// SIMATIC STEP 7 (V5.x) project Daysil_Autoklv_v3_upload
// station: P_ADR_BUS
// station: Hardware
// station: SLIO_CPU_015
// program: S7 Program(1)

FUNCTION_BLOCK FB 1
VERSION : 0.1
BEGIN
// (block stored without names or comments; labels and parameter names are numbered)
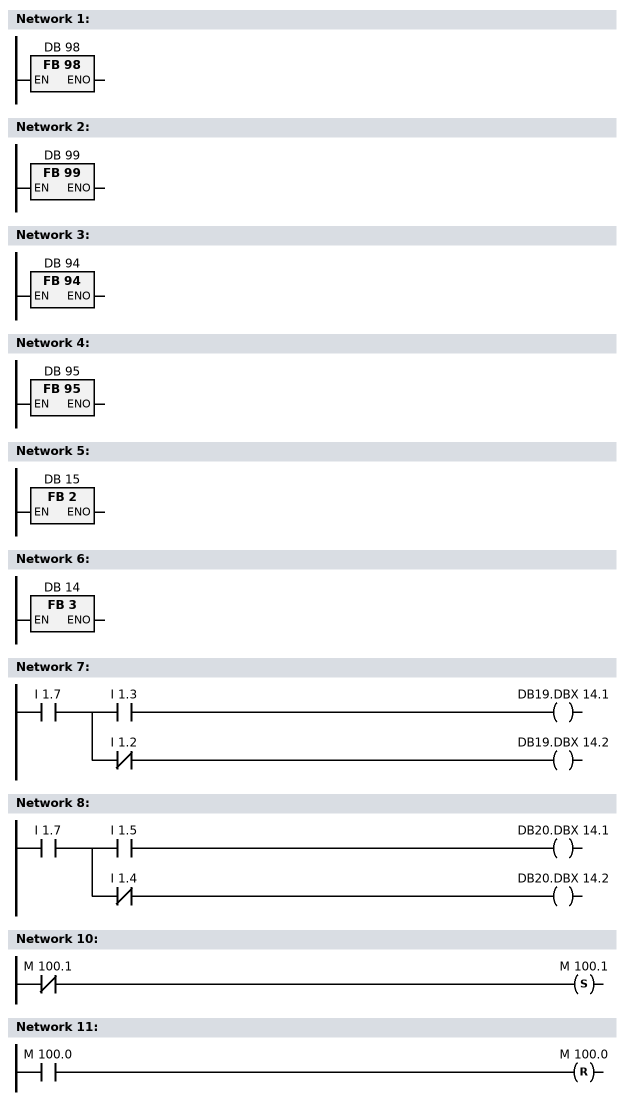
NETWORK
TITLE =
      CALL  FB 98 , DB 98;
      NOP   0;
NETWORK
TITLE =
      CALL  FB 99 , DB 99;
      NOP   0;
NETWORK
TITLE =
      CALL  FB 94 , DB 94;
      NOP   0;
NETWORK
TITLE =
      CALL  FB 95 , DB 95;
      NOP   0;
NETWORK
TITLE =
      CALL  FB 2 , DB 15;
      NOP   0;
NETWORK
TITLE =
      CALL  FB 3 , DB 14;
      NOP   0;
NETWORK
TITLE =
      A     I 1.7;
      =     L 0.0;
      A     L 0.0;
      A     I 1.3;
      =     DB19.DBX 14.1;
      A     L 0.0;
      AN    I 1.2;
      =     DB19.DBX 14.2;
NETWORK
TITLE =
      A     I 1.7;
      =     L 0.0;
      A     L 0.0;
      A     I 1.5;
      =     DB20.DBX 14.1;
      A     L 0.0;
      AN    I 1.4;
      =     DB20.DBX 14.2;
NETWORK
TITLE =
NETWORK
TITLE =
      AN    M 100.1;
      S     M 100.1;
NETWORK
TITLE =
      A     M 100.0;
      R     M 100.0;
NETWORK
TITLE =
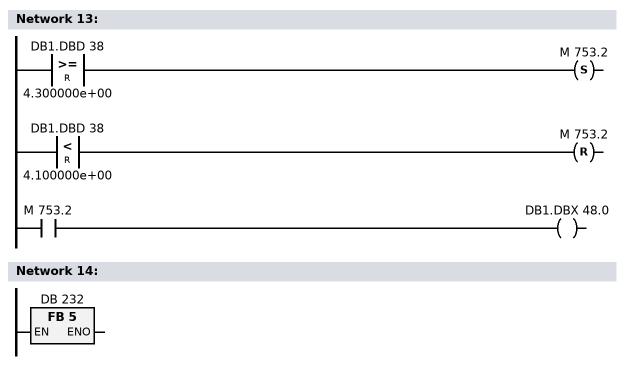
NETWORK
TITLE =
      A(;
      L     DB1.DBD 38;
      L     4.300000e+00;
      >=R;
      );
      S     M 753.2;
      A(;
      L     DB1.DBD 38;
      L     4.100000e+00;
      <R;
      );
      R     M 753.2;
      A     M 753.2;
      =     DB1.DBX 48.0;
NETWORK
TITLE =
      CALL  FB 5 , DB 232;
      NOP   0;
END_FUNCTION_BLOCK

FUNCTION_BLOCK FB 2
VERSION : 0.1
BEGIN
// (block stored without names or comments; labels and parameter names are numbered)
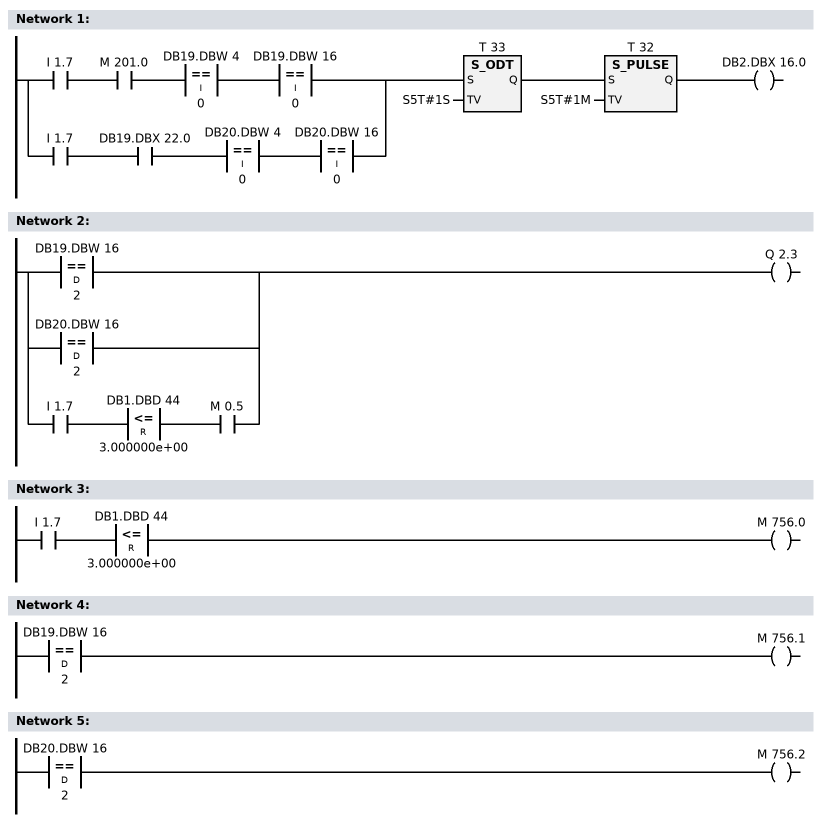
NETWORK
TITLE =
      A(;
      A(;
      A     I 1.7;
      A     M 201.0;
      A(;
      L     DB19.DBW 4;
      L     0;
      ==I;
      );
      A(;
      L     DB19.DBW 16;
      L     0;
      ==I;
      );
      O;
      A     I 1.7;
      A     DB19.DBX 22.0;
      A(;
      L     DB20.DBW 4;
      L     0;
      ==I;
      );
      A(;
      L     DB20.DBW 16;
      L     0;
      ==I;
      );
      );
      L     S5T#1S;
      SD    T 33;
      NOP   0;
      NOP   0;
      NOP   0;
      A     T 33;
      );
      L     S5T#1M;
      SP    T 32;
      NOP   0;
      NOP   0;
      NOP   0;
      A     T 32;
      =     DB2.DBX 16.0;
NETWORK
TITLE =
      O(;
      L     DB19.DBW 16;
      L     2;
      ==D;
      );
      O(;
      L     DB20.DBW 16;
      L     2;
      ==D;
      );
      O;
      A     I 1.7;
      A(;
      L     DB1.DBD 44;
      L     3.000000e+00;
      <=R;
      );
      A     M 0.5;
      =     Q 2.3;
NETWORK
TITLE =
      A     I 1.7;
      A(;
      L     DB1.DBD 44;
      L     3.000000e+00;
      <=R;
      );
      =     M 756.0;
NETWORK
TITLE =
      L     DB19.DBW 16;
      L     2;
      ==D;
      =     M 756.1;
NETWORK
TITLE =
      L     DB20.DBW 16;
      L     2;
      ==D;
      =     M 756.2;
END_FUNCTION_BLOCK

FUNCTION_BLOCK FB 3
VERSION : 0.1
BEGIN
// (block stored without names or comments; labels and parameter names are numbered)
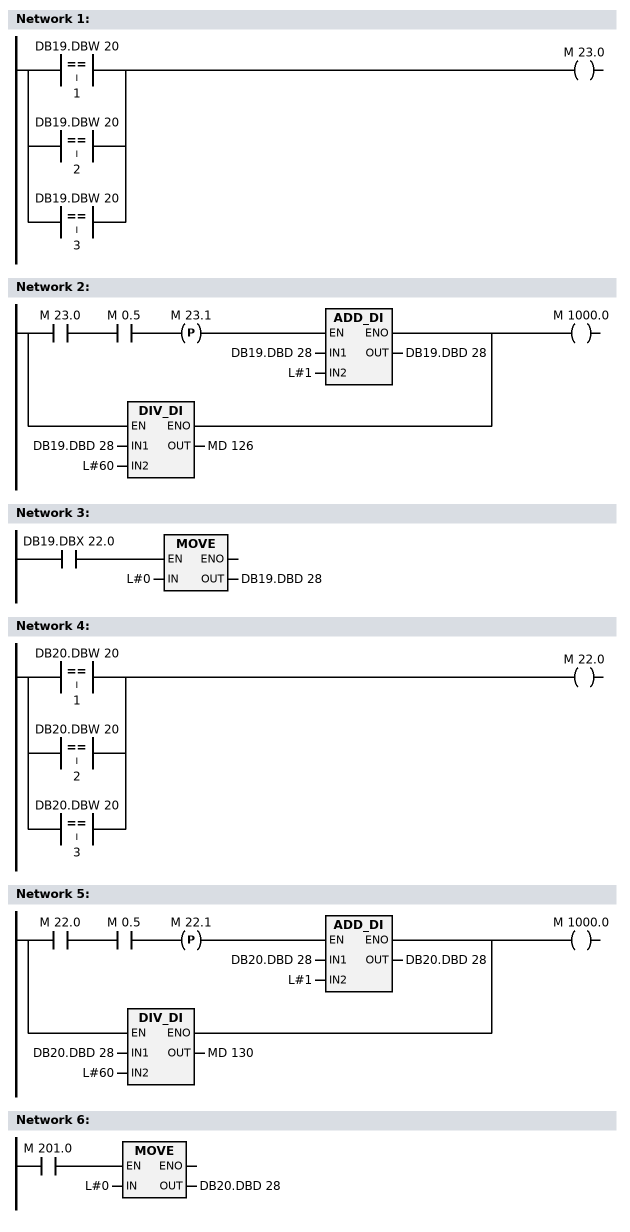
NETWORK
TITLE =
      O(;
      L     DB19.DBW 20;
      L     1;
      ==I;
      );
      O(;
      L     DB19.DBW 20;
      L     2;
      ==I;
      );
      O(;
      L     DB19.DBW 20;
      L     3;
      ==I;
      );
      =     M 23.0;
NETWORK
TITLE =
      O(;
      A     M 23.0;
      A     M 0.5;
      FP    M 23.1;
      JNB   M001;
      L     DB19.DBD 28;
      L     L#1;
      +D;
      T     DB19.DBD 28;
      AN    OV;
      SAVE;
      CLR;
M001: A     BR;
      );
      O(;
      L     DB19.DBD 28;
      L     L#60;
      /D;
      T     MD 126;
      AN    OV;
      SAVE;
      CLR;
      A     BR;
      );
      =     M 1000.0;
NETWORK
TITLE =
      A     DB19.DBX 22.0;
      JNB   M002;
      L     L#0;
      T     DB19.DBD 28;
M002: NOP   0;
NETWORK
TITLE =
      O(;
      L     DB20.DBW 20;
      L     1;
      ==I;
      );
      O(;
      L     DB20.DBW 20;
      L     2;
      ==I;
      );
      O(;
      L     DB20.DBW 20;
      L     3;
      ==I;
      );
      =     M 22.0;
NETWORK
TITLE =
      O(;
      A     M 22.0;
      A     M 0.5;
      FP    M 22.1;
      JNB   M003;
      L     DB20.DBD 28;
      L     L#1;
      +D;
      T     DB20.DBD 28;
      AN    OV;
      SAVE;
      CLR;
M003: A     BR;
      );
      O(;
      L     DB20.DBD 28;
      L     L#60;
      /D;
      T     MD 130;
      AN    OV;
      SAVE;
      CLR;
      A     BR;
      );
      =     M 1000.0;
NETWORK
TITLE =
      A     M 201.0;
      JNB   M004;
      L     L#0;
      T     DB20.DBD 28;
M004: NOP   0;
NETWORK
TITLE =
      O(;
      A(;
      A     DB17.DBX 40.3;
      =     L 0.0;
      BLD   103;
      BLD   9;
      =     L 5.0;
      CDB;
      OPN   DI 5;
      TAR2  LD 1;
      A     L 0.0;
      =     DIX 0.0;
      L     L#82800000;
      T     DID 2;
      LAR2  P#DBX 0.0;
      UC    SFB 4;
      LAR2  LD 1;
      L     DID 8;
      OPN   DI 17;
      T     DID 42;
      OPN   DI 5;
      CDB;
      BLD   10;
      A     BR;
      );
      JNB   M005;
      CALL  FC 1 (
           $1                       := DB17.DBD 42,
           $2                       := DB17.DBW 4,
           $3                       := DB17.DBD 46);
M005: A     BR;
      );
      O(;
      L     DB17.DBD 46;
      L     60;
      /D;
      T     MD 118;
      AN    OV;
      SAVE;
      CLR;
      A     BR;
      );
      =     M 1000.0;
NETWORK
TITLE =
      O(;
      A(;
      A     DB18.DBX 40.3;
      =     L 0.0;
      BLD   103;
      BLD   9;
      =     L 5.0;
      CDB;
      OPN   DI 6;
      TAR2  LD 1;
      A     L 0.0;
      =     DIX 0.0;
      L     L#82800000;
      T     DID 2;
      LAR2  P#DBX 0.0;
      UC    SFB 4;
      LAR2  LD 1;
      L     DID 8;
      OPN   DI 18;
      T     DID 42;
      OPN   DI 6;
      CDB;
      BLD   10;
      A     BR;
      );
      JNB   M006;
      CALL  FC 1 (
           $1                       := DB18.DBD 42,
           $2                       := DB18.DBW 4,
           $3                       := DB18.DBD 46);
M006: A     BR;
      );
      O(;
      L     DB18.DBD 46;
      L     60;
      /D;
      T     MD 122;
      AN    OV;
      SAVE;
      CLR;
      A     BR;
      );
      =     M 1000.0;
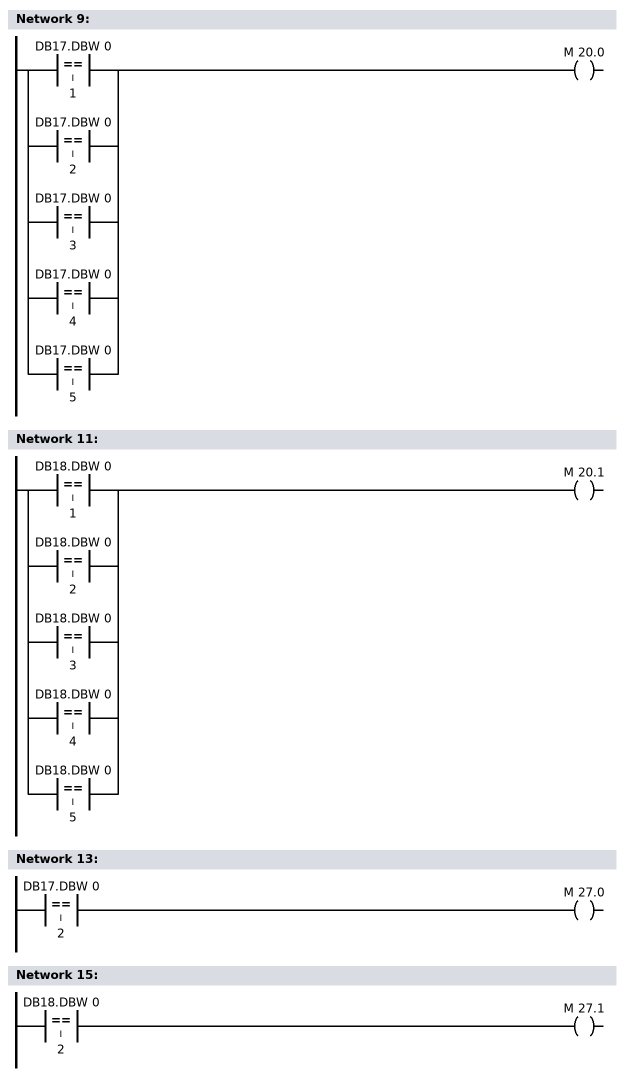
NETWORK
TITLE =
      O(;
      L     DB17.DBW 0;
      L     1;
      ==I;
      );
      O(;
      L     DB17.DBW 0;
      L     2;
      ==I;
      );
      O(;
      L     DB17.DBW 0;
      L     3;
      ==I;
      );
      O(;
      L     DB17.DBW 0;
      L     4;
      ==I;
      );
      O(;
      L     DB17.DBW 0;
      L     5;
      ==I;
      );
      =     M 20.0;
NETWORK
TITLE =
      O(;
      A(;
      A     M 20.0;
      =     L 0.0;
      BLD   103;
      BLD   9;
      =     L 5.0;
      CDB;
      OPN   DI 7;
      TAR2  LD 1;
      A     L 0.0;
      =     DIX 0.0;
      L     L#82800000;
      T     DID 2;
      LAR2  P#DBX 0.0;
      UC    SFB 4;
      LAR2  LD 1;
      L     DID 8;
      OPN   DI 17;
      T     DID 50;
      OPN   DI 7;
      CDB;
      BLD   10;
      A     BR;
      );
      JNB   M007;
      L     DB17.DBD 50;
      L     1000;
      /D;
      T     DB17.DBD 54;
      AN    OV;
      SAVE;
      CLR;
M007: A     BR;
      );
      O(;
      L     DB17.DBD 54;
      L     60;
      /D;
      T     MD 110;
      AN    OV;
      SAVE;
      CLR;
      A     BR;
      );
      =     M 1000.0;
NETWORK
TITLE =
      O(;
      L     DB18.DBW 0;
      L     1;
      ==I;
      );
      O(;
      L     DB18.DBW 0;
      L     2;
      ==I;
      );
      O(;
      L     DB18.DBW 0;
      L     3;
      ==I;
      );
      O(;
      L     DB18.DBW 0;
      L     4;
      ==I;
      );
      O(;
      L     DB18.DBW 0;
      L     5;
      ==I;
      );
      =     M 20.1;
NETWORK
TITLE =
      O(;
      A(;
      A     M 20.1;
      =     L 0.0;
      BLD   103;
      BLD   9;
      =     L 5.0;
      CDB;
      OPN   DI 8;
      TAR2  LD 1;
      A     L 0.0;
      =     DIX 0.0;
      L     L#82800000;
      T     DID 2;
      LAR2  P#DBX 0.0;
      UC    SFB 4;
      LAR2  LD 1;
      L     DID 8;
      OPN   DI 18;
      T     DID 50;
      OPN   DI 8;
      CDB;
      BLD   10;
      A     BR;
      );
      JNB   M008;
      L     DB18.DBD 50;
      L     1000;
      /D;
      T     DB18.DBD 54;
      AN    OV;
      SAVE;
      CLR;
M008: A     BR;
      );
      O(;
      L     DB18.DBD 54;
      L     60;
      /D;
      T     MD 114;
      AN    OV;
      SAVE;
      CLR;
      A     BR;
      );
      =     M 1000.0;
NETWORK
TITLE =
      L     DB17.DBW 0;
      L     2;
      ==I;
      =     M 27.0;
NETWORK
TITLE =
      A(;
      A     M 27.0;
      =     L 0.0;
      BLD   103;
      BLD   9;
      =     L 5.0;
      CDB;
      OPN   DI 9;
      TAR2  LD 1;
      A     L 0.0;
      =     DIX 0.0;
      L     L#82800000;
      T     DID 2;
      LAR2  P#DBX 0.0;
      UC    SFB 4;
      LAR2  LD 1;
      L     DID 8;
      OPN   DI 17;
      T     DID 58;
      OPN   DI 9;
      CDB;
      BLD   10;
      A     BR;
      );
      JNB   M009;
      L     DB17.DBD 58;
      L     1000;
      /D;
      T     DB17.DBD 62;
M009: NOP   0;
NETWORK
TITLE =
      L     DB18.DBW 0;
      L     2;
      ==I;
      =     M 27.1;
NETWORK
TITLE =
      A(;
      A     M 27.1;
      =     L 0.0;
      BLD   103;
      BLD   9;
      =     L 5.0;
      CDB;
      OPN   DI 10;
      TAR2  LD 1;
      A     L 0.0;
      =     DIX 0.0;
      L     L#82800000;
      T     DID 2;
      LAR2  P#DBX 0.0;
      UC    SFB 4;
      LAR2  LD 1;
      L     DID 8;
      OPN   DI 18;
      T     DID 58;
      OPN   DI 10;
      CDB;
      BLD   10;
      A     BR;
      );
      JNB   M010;
      L     DB18.DBD 58;
      L     1000;
      /D;
      T     DB18.DBD 62;
M010: NOP   0;
END_FUNCTION_BLOCK

FUNCTION_BLOCK FB 5
VERSION : 0.1
BEGIN
// (block stored without names or comments; labels and parameter names are numbered)
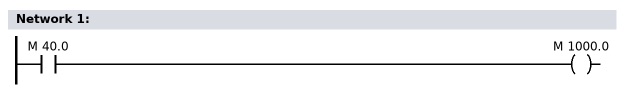
NETWORK
TITLE =
      A     M 40.0;
      =     M 1000.0;
END_FUNCTION_BLOCK

FUNCTION_BLOCK FB 20
VERSION : 0.1
BEGIN
// (block stored without names or comments; labels and parameter names are numbered)
NETWORK
TITLE =
      A(;
      A(;
      A     M 100.0;
      =     L 0.0;
      BLD   103;
      CALL  FC 105 (
           $1                       := DIW [AR2,P#4.0],
           $2                       := DID [AR2,P#24.0],
           $3                       := DID [AR2,P#28.0],
           $4                       := L 0.0,
           $5                       := DIW [AR2,P#116.0],
           $6                       := DID [AR2,P#118.0]);
      A     BR;
      );
      JNB   M001;
      L     DIW [AR2,P#116.0];
      T     DIW [AR2,P#68.0];
      SET;
      SAVE;
      CLR;
M001: A     BR;
      );
      JNB   M002;
      L     DID [AR2,P#118.0];
      T     DID [AR2,P#70.0];
M002: NOP   0;
NETWORK
TITLE =
      A(;
      A(;
      A     M 100.0;
      =     L 0.0;
      BLD   103;
      CALL  FC 105 (
           $1                       := DIW [AR2,P#40.0],
           $2                       := DID [AR2,P#32.0],
           $3                       := DID [AR2,P#36.0],
           $4                       := L 0.0,
           $5                       := DIW [AR2,P#122.0],
           $6                       := DID [AR2,P#124.0]);
      A     BR;
      );
      JNB   M003;
      L     DIW [AR2,P#122.0];
      T     DIW [AR2,P#76.0];
      SET;
      SAVE;
      CLR;
M003: A     BR;
      );
      JNB   M004;
      L     DID [AR2,P#124.0];
      T     DID [AR2,P#78.0];
M004: NOP   0;
NETWORK
TITLE =
      A(;
      A     I 1.7;
      A     DIX [AR2,P#0.0];
      A     DB1.DBX 48.0;
      L     S5T#200MS;
      T     LD 0;
      TAK;
      T     LD 4;
      L     DIW [AR2,P#14.0];
      T     LW 8;
      L     LD 4;
      L     LD 0;
      SD    T [LW 8];
      NOP   0;
      NOP   0;
      NOP   0;
      T     LD 0;
      TAK;
      T     LD 4;
      L     DIW [AR2,P#14.0];
      T     LW 8;
      L     LD 4;
      L     LD 0;
      A     T [LW 8];
      );
      A     DIX [AR2,P#0.4];
      A     DIX [AR2,P#0.1];
      A(;
      L     DIW [AR2,P#84.0];
      L     0;
      ==I;
      );
      JNB   M005;
      L     1;
      T     DIW [AR2,P#84.0];
      SET;
      SAVE;
      CLR;
M005: A     BR;
      S     DIX [AR2,P#128.0];
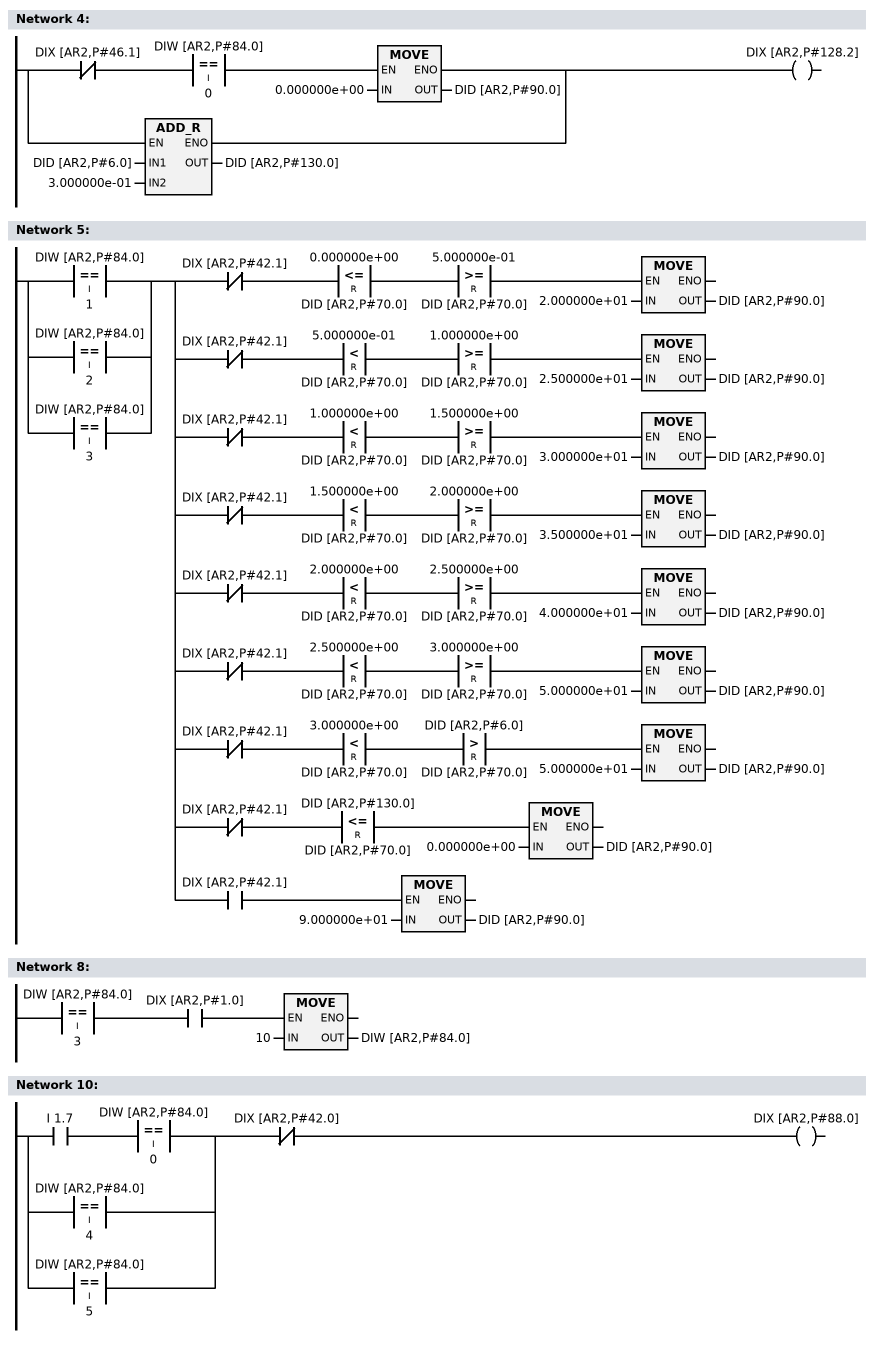
NETWORK
TITLE =
      O(;
      AN    DIX [AR2,P#46.1];
      A(;
      L     DIW [AR2,P#84.0];
      L     0;
      ==I;
      );
      JNB   M006;
      L     0.000000e+00;
      T     DID [AR2,P#90.0];
      SET;
      SAVE;
      CLR;
M006: A     BR;
      );
      O(;
      L     DID [AR2,P#6.0];
      L     3.000000e-01;
      +R;
      T     DID [AR2,P#130.0];
      AN    OV;
      SAVE;
      CLR;
      A     BR;
      );
      =     DIX [AR2,P#128.2];
NETWORK
TITLE =
      O(;
      L     DIW [AR2,P#84.0];
      L     1;
      ==I;
      );
      O(;
      L     DIW [AR2,P#84.0];
      L     2;
      ==I;
      );
      O(;
      L     DIW [AR2,P#84.0];
      L     3;
      ==I;
      );
      =     L 0.0;
      A     L 0.0;
      AN    DIX [AR2,P#42.1];
      A(;
      L     0.000000e+00;
      L     DID [AR2,P#70.0];
      <=R;
      );
      A(;
      L     5.000000e-01;
      L     DID [AR2,P#70.0];
      >=R;
      );
      JNB   M007;
      L     2.000000e+01;
      T     DID [AR2,P#90.0];
M007: NOP   0;
      A     L 0.0;
      AN    DIX [AR2,P#42.1];
      A(;
      L     5.000000e-01;
      L     DID [AR2,P#70.0];
      <R;
      );
      A(;
      L     1.000000e+00;
      L     DID [AR2,P#70.0];
      >=R;
      );
      JNB   M008;
      L     2.500000e+01;
      T     DID [AR2,P#90.0];
M008: NOP   0;
      A     L 0.0;
      AN    DIX [AR2,P#42.1];
      A(;
      L     1.000000e+00;
      L     DID [AR2,P#70.0];
      <R;
      );
      A(;
      L     1.500000e+00;
      L     DID [AR2,P#70.0];
      >=R;
      );
      JNB   M009;
      L     3.000000e+01;
      T     DID [AR2,P#90.0];
M009: NOP   0;
      A     L 0.0;
      AN    DIX [AR2,P#42.1];
      A(;
      L     1.500000e+00;
      L     DID [AR2,P#70.0];
      <R;
      );
      A(;
      L     2.000000e+00;
      L     DID [AR2,P#70.0];
      >=R;
      );
      JNB   M010;
      L     3.500000e+01;
      T     DID [AR2,P#90.0];
M010: NOP   0;
      A     L 0.0;
      AN    DIX [AR2,P#42.1];
      A(;
      L     2.000000e+00;
      L     DID [AR2,P#70.0];
      <R;
      );
      A(;
      L     2.500000e+00;
      L     DID [AR2,P#70.0];
      >=R;
      );
      JNB   M011;
      L     4.000000e+01;
      T     DID [AR2,P#90.0];
M011: NOP   0;
      A     L 0.0;
      AN    DIX [AR2,P#42.1];
      A(;
      L     2.500000e+00;
      L     DID [AR2,P#70.0];
      <R;
      );
      A(;
      L     3.000000e+00;
      L     DID [AR2,P#70.0];
      >=R;
      );
      JNB   M012;
      L     5.000000e+01;
      T     DID [AR2,P#90.0];
M012: NOP   0;
      A     L 0.0;
      AN    DIX [AR2,P#42.1];
      A(;
      L     3.000000e+00;
      L     DID [AR2,P#70.0];
      <R;
      );
      A(;
      L     DID [AR2,P#6.0];
      L     DID [AR2,P#70.0];
      >R;
      );
      JNB   M013;
      L     5.000000e+01;
      T     DID [AR2,P#90.0];
M013: NOP   0;
      A     L 0.0;
      AN    DIX [AR2,P#42.1];
      A(;
      L     DID [AR2,P#130.0];
      L     DID [AR2,P#70.0];
      <=R;
      );
      JNB   M014;
      L     0.000000e+00;
      T     DID [AR2,P#90.0];
M014: NOP   0;
      A     L 0.0;
      A     DIX [AR2,P#42.1];
      JNB   M015;
      L     9.000000e+01;
      T     DID [AR2,P#90.0];
M015: NOP   0;
NETWORK
TITLE =
      L     DIW [AR2,P#84.0];
      L     1;
      ==I;
      =     L 0.0;
      A(;
      A     L 0.0;
      A     DIX [AR2,P#104.0];
      L     DIW [AR2,P#2.0];
      T     LD 1;
      TAK;
      T     LD 5;
      L     DIW [AR2,P#18.0];
      T     LW 9;
      L     LD 5;
      L     LD 1;
      SD    T [LW 9];
      NOP   0;
      NOP   0;
      NOP   0;
      T     LD 1;
      TAK;
      T     LD 5;
      L     DIW [AR2,P#18.0];
      T     LW 9;
      L     LD 5;
      L     LD 1;
      A     T [LW 9];
      );
      JNB   M016;
      L     2;
      T     DIW [AR2,P#84.0];
M016: NOP   0;
      A     L 0.0;
      A(;
      O(;
      L     DID [AR2,P#70.0];
      L     DID [AR2,P#6.0];
      >=R;
      );
      O     DIX [AR2,P#104.0];
      );
      =     DIX [AR2,P#104.0];
NETWORK
TITLE =
      L     DIW [AR2,P#84.0];
      L     2;
      ==I;
      =     L 0.0;
      A     L 0.0;
      L     S5T#5M;
      T     LD 1;
      TAK;
      T     LD 5;
      L     DIW [AR2,P#56.0];
      T     LW 9;
      L     LD 5;
      L     LD 1;
      SD    T [LW 9];
      NOP   0;
      NOP   0;
      NOP   0;
      NOP   0;
      A     L 0.0;
      A     DIX [AR2,P#0.2];
      JNB   M017;
      L     3;
      T     DIW [AR2,P#84.0];
M017: NOP   0;
      A     L 0.0;
      A     DIX [AR2,P#0.3];
      JNB   M018;
      L     4;
      T     DIW [AR2,P#84.0];
M018: NOP   0;
NETWORK
TITLE =
      A(;
      L     DIW [AR2,P#84.0];
      L     3;
      ==I;
      );
      A     DIX [AR2,P#1.0];
      JNB   M019;
      L     10;
      T     DIW [AR2,P#84.0];
M019: NOP   0;
NETWORK
TITLE =
      L     DIW [AR2,P#84.0];
      L     10;
      ==I;
      =     L 0.0;
      A     L 0.0;
      JNB   M020;
      L     9.000000e+01;
      T     DID [AR2,P#90.0];
      SET;
      SAVE;
      CLR;
M020: A     BR;
      =     DIX [AR2,P#66.0];
      A(;
      A     L 0.0;
      L     S5T#23S;
      T     LD 1;
      TAK;
      T     LD 5;
      L     DIW [AR2,P#20.0];
      T     LW 9;
      L     LD 5;
      L     LD 1;
      SD    T [LW 9];
      NOP   0;
      NOP   0;
      NOP   0;
      T     LD 1;
      TAK;
      T     LD 5;
      L     DIW [AR2,P#20.0];
      T     LW 9;
      L     LD 5;
      L     LD 1;
      A     T [LW 9];
      );
      JNB   M021;
      L     4;
      T     DIW [AR2,P#84.0];
M021: NOP   0;
NETWORK
TITLE =
      A(;
      A     I 1.7;
      A(;
      L     DIW [AR2,P#84.0];
      L     0;
      ==I;
      );
      O(;
      L     DIW [AR2,P#84.0];
      L     4;
      ==I;
      );
      O(;
      L     DIW [AR2,P#84.0];
      L     5;
      ==I;
      );
      );
      AN    DIX [AR2,P#42.0];
      =     DIX [AR2,P#88.0];
NETWORK
TITLE =
      L     DIW [AR2,P#84.0];
      L     4;
      ==I;
      =     L 0.0;
      A     L 0.0;
      JNB   M022;
      L     0.000000e+00;
      T     DID [AR2,P#90.0];
M022: NOP   0;
      A     L 0.0;
      BLD   102;
      =     DIX [AR2,P#128.1];
      A     L 0.0;
      A(;
      L     DID [AR2,P#70.0];
      L     1.000000e-01;
      <=R;
      );
      =     L 0.1;
      A     L 0.1;
      BLD   102;
      S     DIX [AR2,P#114.1];
      A(;
      A     L 0.1;
      L     S5T#5S;
      T     LD 1;
      TAK;
      T     LD 5;
      L     DIW [AR2,P#52.0];
      T     LW 9;
      L     LD 5;
      L     LD 1;
      SD    T [LW 9];
      NOP   0;
      NOP   0;
      NOP   0;
      T     LD 1;
      TAK;
      T     LD 5;
      L     DIW [AR2,P#52.0];
      T     LW 9;
      L     LD 5;
      L     LD 1;
      A     T [LW 9];
      );
      JNB   M023;
      L     5;
      T     DIW [AR2,P#84.0];
M023: NOP   0;
NETWORK
TITLE =
      A(;
      A(;
      L     DIW [AR2,P#84.0];
      L     5;
      ==I;
      );
      L     S5T#1S;
      T     LD 0;
      TAK;
      T     LD 4;
      L     DIW [AR2,P#54.0];
      T     LW 8;
      L     LD 4;
      L     LD 0;
      SD    T [LW 8];
      NOP   0;
      NOP   0;
      NOP   0;
      T     LD 0;
      TAK;
      T     LD 4;
      L     DIW [AR2,P#54.0];
      T     LW 8;
      L     LD 4;
      L     LD 0;
      A     T [LW 8];
      );
      AN    DIX [AR2,P#0.4];
      JNB   M024;
      L     0;
      T     DIW [AR2,P#84.0];
M024: NOP   0;
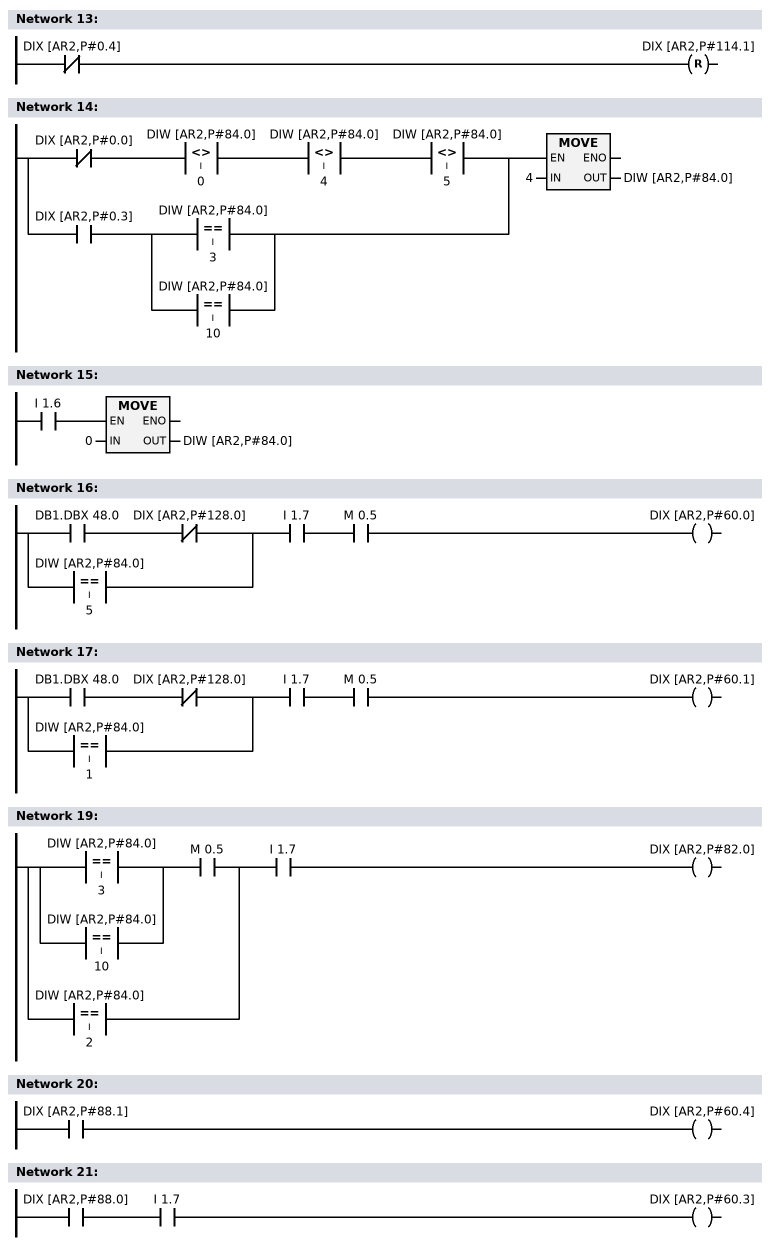
NETWORK
TITLE =
      AN    DIX [AR2,P#0.4];
      R     DIX [AR2,P#114.1];
NETWORK
TITLE =
      A(;
      AN    DIX [AR2,P#0.0];
      A(;
      L     DIW [AR2,P#84.0];
      L     0;
      <>I;
      );
      A(;
      L     DIW [AR2,P#84.0];
      L     4;
      <>I;
      );
      A(;
      L     DIW [AR2,P#84.0];
      L     5;
      <>I;
      );
      O;
      A     DIX [AR2,P#0.3];
      A(;
      O(;
      L     DIW [AR2,P#84.0];
      L     3;
      ==I;
      );
      O(;
      L     DIW [AR2,P#84.0];
      L     10;
      ==I;
      );
      );
      );
      JNB   M025;
      L     4;
      T     DIW [AR2,P#84.0];
M025: NOP   0;
NETWORK
TITLE =
      A     I 1.6;
      JNB   M026;
      L     0;
      T     DIW [AR2,P#84.0];
M026: NOP   0;
NETWORK
TITLE =
      A(;
      A     DB1.DBX 48.0;
      AN    DIX [AR2,P#128.0];
      O(;
      L     DIW [AR2,P#84.0];
      L     5;
      ==I;
      );
      );
      A     I 1.7;
      A     M 0.5;
      =     DIX [AR2,P#60.0];
NETWORK
TITLE =
      A(;
      A     DB1.DBX 48.0;
      AN    DIX [AR2,P#128.0];
      O(;
      L     DIW [AR2,P#84.0];
      L     1;
      ==I;
      );
      );
      A     I 1.7;
      A     M 0.5;
      =     DIX [AR2,P#60.1];
NETWORK
TITLE =
      A(;
      A(;
      L     DIW [AR2,P#84.0];
      L     2;
      ==I;
      );
      A     M 0.5;
      O(;
      A(;
      O(;
      L     DIW [AR2,P#84.0];
      L     3;
      ==I;
      );
      O(;
      L     DIW [AR2,P#84.0];
      L     10;
      ==I;
      );
      );
      AN    DIX [AR2,P#66.0];
      L     S5T#5M;
      T     LD 0;
      TAK;
      T     LD 4;
      L     DIW [AR2,P#58.0];
      T     LW 8;
      L     LD 4;
      L     LD 0;
      SD    T [LW 8];
      NOP   0;
      NOP   0;
      NOP   0;
      T     LD 0;
      TAK;
      T     LD 4;
      L     DIW [AR2,P#58.0];
      T     LW 8;
      L     LD 4;
      L     LD 0;
      A     T [LW 8];
      );
      );
      A     I 1.7;
      =     DIX [AR2,P#60.2];
NETWORK
TITLE =
      A(;
      A(;
      O(;
      L     DIW [AR2,P#84.0];
      L     3;
      ==I;
      );
      O(;
      L     DIW [AR2,P#84.0];
      L     10;
      ==I;
      );
      );
      A     M 0.5;
      O(;
      L     DIW [AR2,P#84.0];
      L     2;
      ==I;
      );
      );
      A     I 1.7;
      =     DIX [AR2,P#82.0];
NETWORK
TITLE =
      A     DIX [AR2,P#88.1];
      =     DIX [AR2,P#60.4];
NETWORK
TITLE =
      A     DIX [AR2,P#88.0];
      A     I 1.7;
      =     DIX [AR2,P#60.3];
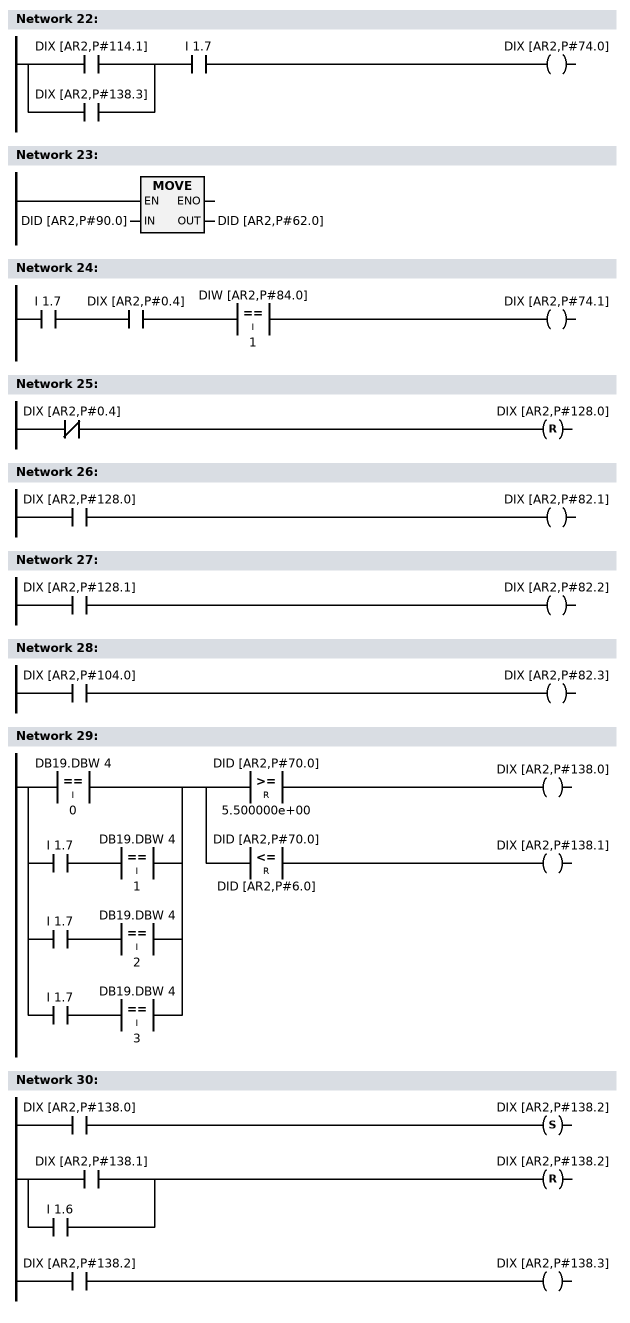
NETWORK
TITLE =
      A(;
      O     DIX [AR2,P#114.1];
      O     DIX [AR2,P#138.3];
      );
      A     I 1.7;
      =     DIX [AR2,P#74.0];
NETWORK
TITLE =
      L     DID [AR2,P#90.0];
      T     DID [AR2,P#62.0];
      NOP   0;
NETWORK
TITLE =
      A     I 1.7;
      A     DIX [AR2,P#0.4];
      A(;
      L     DIW [AR2,P#84.0];
      L     1;
      ==I;
      );
      =     DIX [AR2,P#74.1];
NETWORK
TITLE =
      AN    DIX [AR2,P#0.4];
      R     DIX [AR2,P#128.0];
NETWORK
TITLE =
      A     DIX [AR2,P#128.0];
      =     DIX [AR2,P#82.1];
NETWORK
TITLE =
      A     DIX [AR2,P#128.1];
      =     DIX [AR2,P#82.2];
NETWORK
TITLE =
      A     DIX [AR2,P#104.0];
      =     DIX [AR2,P#82.3];
NETWORK
TITLE =
      O(;
      L     DB19.DBW 4;
      L     0;
      ==I;
      );
      O;
      A     I 1.7;
      A(;
      L     DB19.DBW 4;
      L     1;
      ==I;
      );
      O;
      A     I 1.7;
      A(;
      L     DB19.DBW 4;
      L     2;
      ==I;
      );
      O;
      A     I 1.7;
      A(;
      L     DB19.DBW 4;
      L     3;
      ==I;
      );
      =     L 0.0;
      A     L 0.0;
      A(;
      L     DID [AR2,P#70.0];
      L     5.500000e+00;
      >=R;
      );
      =     DIX [AR2,P#138.0];
      A     L 0.0;
      A(;
      L     DID [AR2,P#70.0];
      L     DID [AR2,P#6.0];
      <=R;
      );
      =     DIX [AR2,P#138.1];
NETWORK
TITLE =
      A     DIX [AR2,P#138.0];
      S     DIX [AR2,P#138.2];
      A(;
      O     DIX [AR2,P#138.1];
      O     I 1.6;
      );
      R     DIX [AR2,P#138.2];
      A     DIX [AR2,P#138.2];
      =     DIX [AR2,P#138.3];
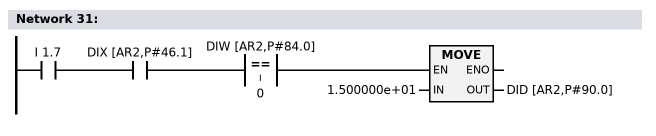
NETWORK
TITLE =
      A     I 1.7;
      A     DIX [AR2,P#46.1];
      A(;
      L     DIW [AR2,P#84.0];
      L     0;
      ==I;
      );
      JNB   M027;
      L     1.500000e+01;
      T     DID [AR2,P#90.0];
M027: NOP   0;
END_FUNCTION_BLOCK

// FB 41: know-how protected block, not included

FUNCTION_BLOCK FB 47
VERSION : 0.1
BEGIN
// (block stored without names or comments; labels and parameter names are numbered)
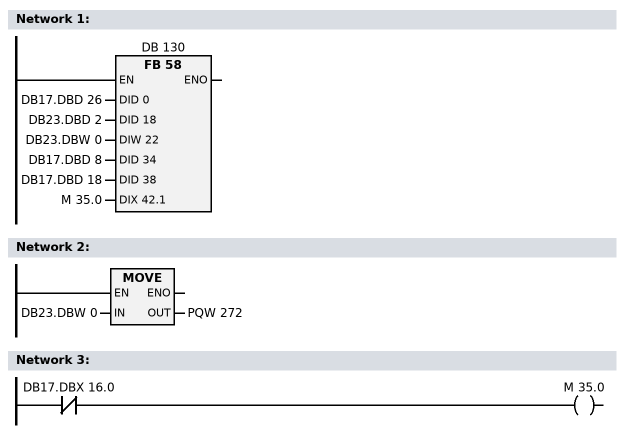
NETWORK
TITLE =
      CALL  FB 58 , DB 130 (
           DID 0                    := DB17.DBD 26,
           DID 18                   := DB23.DBD 2,
           DIW 22                   := DB23.DBW 0,
           DID 34                   := DB17.DBD 8,
           DID 38                   := DB17.DBD 18,
           DIX 42.1                 := M 35.0);
      NOP   0;
NETWORK
TITLE =
      L     DB23.DBW 0;
      T     PQW 272;
      NOP   0;
NETWORK
TITLE =
      AN    DB17.DBX 16.0;
      =     M 35.0;
NETWORK
TITLE =
END_FUNCTION_BLOCK

FUNCTION_BLOCK FB 48
VERSION : 0.1
BEGIN
// (block stored without names or comments; labels and parameter names are numbered)
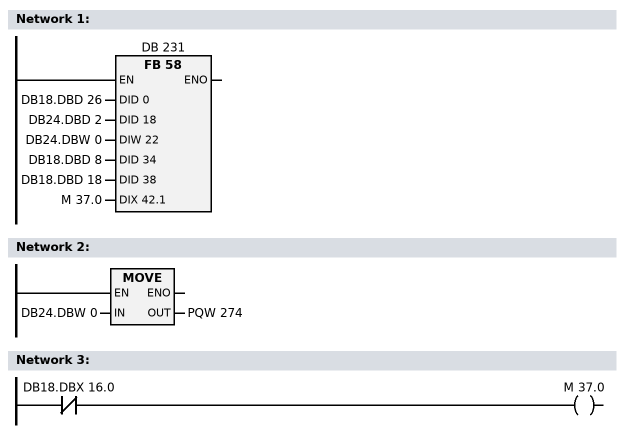
NETWORK
TITLE =
      CALL  FB 58 , DB 231 (
           DID 0                    := DB18.DBD 26,
           DID 18                   := DB24.DBD 2,
           DIW 22                   := DB24.DBW 0,
           DID 34                   := DB18.DBD 8,
           DID 38                   := DB18.DBD 18,
           DIX 42.1                 := M 37.0);
      NOP   0;
NETWORK
TITLE =
      L     DB24.DBW 0;
      T     PQW 274;
      NOP   0;
NETWORK
TITLE =
      AN    DB18.DBX 16.0;
      =     M 37.0;
END_FUNCTION_BLOCK

FUNCTION_BLOCK FB 49
VERSION : 0.1
BEGIN
// (block stored without names or comments; labels and parameter names are numbered)
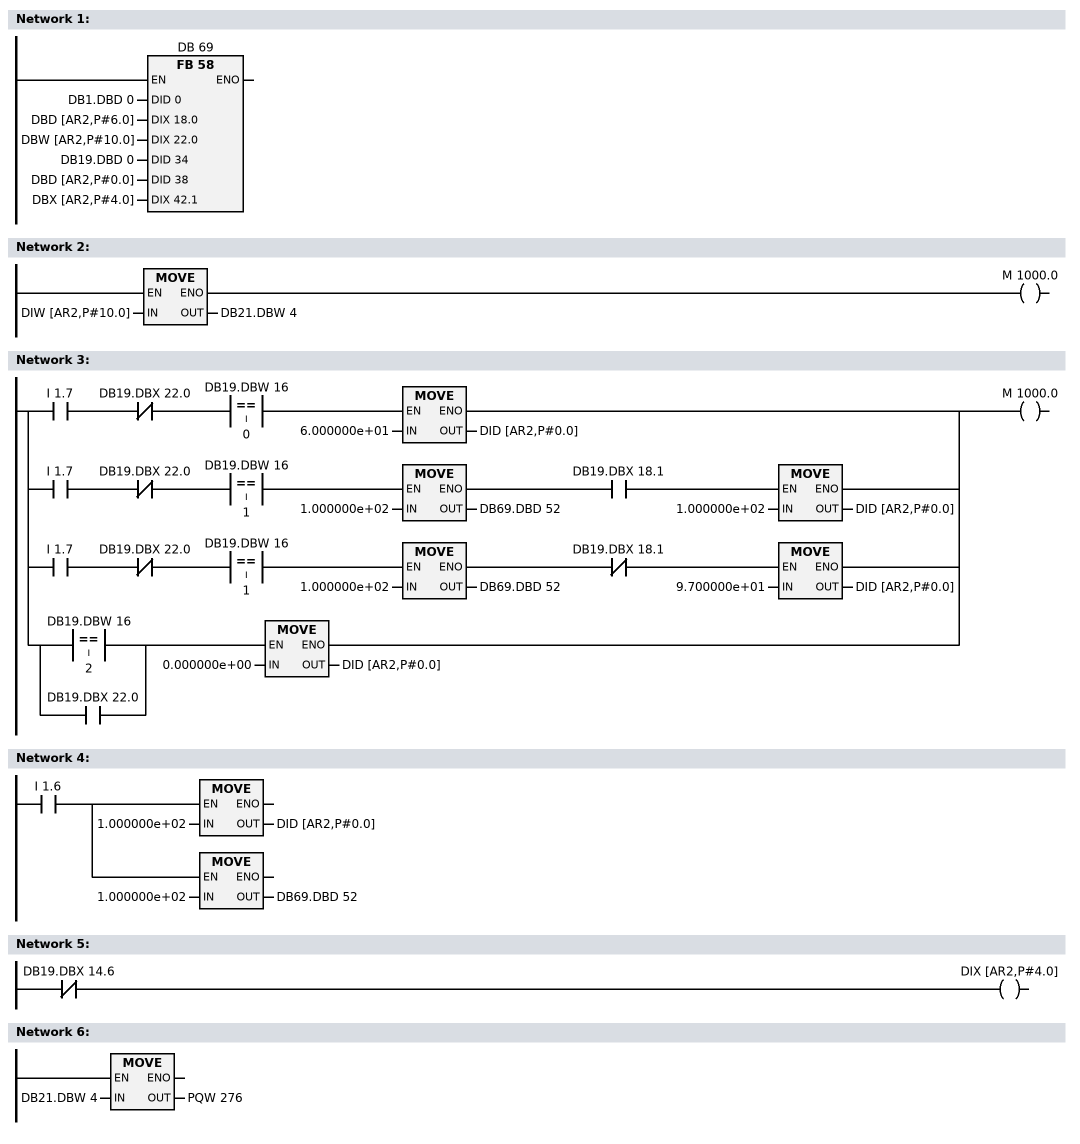
NETWORK
TITLE =
      CALL  FB 58 , DB 69 (
           DID 0                    := DB1.DBD 0,
           DIX 18.0                 := DBD [AR2,P#6.0],
           DIX 22.0                 := DBW [AR2,P#10.0],
           DID 34                   := DB19.DBD 0,
           DID 38                   := DBD [AR2,P#0.0],
           DIX 42.1                 := DBX [AR2,P#4.0]);
      NOP   0;
NETWORK
TITLE =
      L     DIW [AR2,P#10.0];
      T     DB21.DBW 4;
      SET;
      SAVE;
      CLR;
      A     BR;
      =     M 1000.0;
NETWORK
TITLE =
      O(;
      A     I 1.7;
      AN    DB19.DBX 22.0;
      A(;
      L     DB19.DBW 16;
      L     0;
      ==I;
      );
      JNB   M001;
      L     6.000000e+01;
      T     DID [AR2,P#0.0];
      SET;
      SAVE;
      CLR;
M001: A     BR;
      );
      O(;
      A(;
      A     I 1.7;
      AN    DB19.DBX 22.0;
      A(;
      L     DB19.DBW 16;
      L     1;
      ==I;
      );
      JNB   M002;
      L     1.000000e+02;
      T     DB69.DBD 52;
      SET;
      SAVE;
      CLR;
M002: A     BR;
      );
      A     DB19.DBX 18.1;
      JNB   M003;
      L     1.000000e+02;
      T     DID [AR2,P#0.0];
      SET;
      SAVE;
      CLR;
M003: A     BR;
      );
      O(;
      A(;
      A     I 1.7;
      AN    DB19.DBX 22.0;
      A(;
      L     DB19.DBW 16;
      L     1;
      ==I;
      );
      JNB   M004;
      L     1.000000e+02;
      T     DB69.DBD 52;
      SET;
      SAVE;
      CLR;
M004: A     BR;
      );
      AN    DB19.DBX 18.1;
      JNB   M005;
      L     9.700000e+01;
      T     DID [AR2,P#0.0];
      SET;
      SAVE;
      CLR;
M005: A     BR;
      );
      O(;
      A(;
      O(;
      L     DB19.DBW 16;
      L     2;
      ==I;
      );
      O     DB19.DBX 22.0;
      );
      JNB   M006;
      L     0.000000e+00;
      T     DID [AR2,P#0.0];
      SET;
      SAVE;
      CLR;
M006: A     BR;
      );
      =     M 1000.0;
NETWORK
TITLE =
      A     I 1.6;
      =     L 0.0;
      A     L 0.0;
      JNB   M007;
      L     1.000000e+02;
      T     DID [AR2,P#0.0];
M007: NOP   0;
      A     L 0.0;
      JNB   M008;
      L     1.000000e+02;
      T     DB69.DBD 52;
M008: NOP   0;
NETWORK
TITLE =
      AN    DB19.DBX 14.6;
      =     DIX [AR2,P#4.0];
NETWORK
TITLE =
      L     DB21.DBW 4;
      T     PQW 276;
      NOP   0;
END_FUNCTION_BLOCK

FUNCTION_BLOCK FB 50
VERSION : 0.1
BEGIN
// (block stored without names or comments; labels and parameter names are numbered)
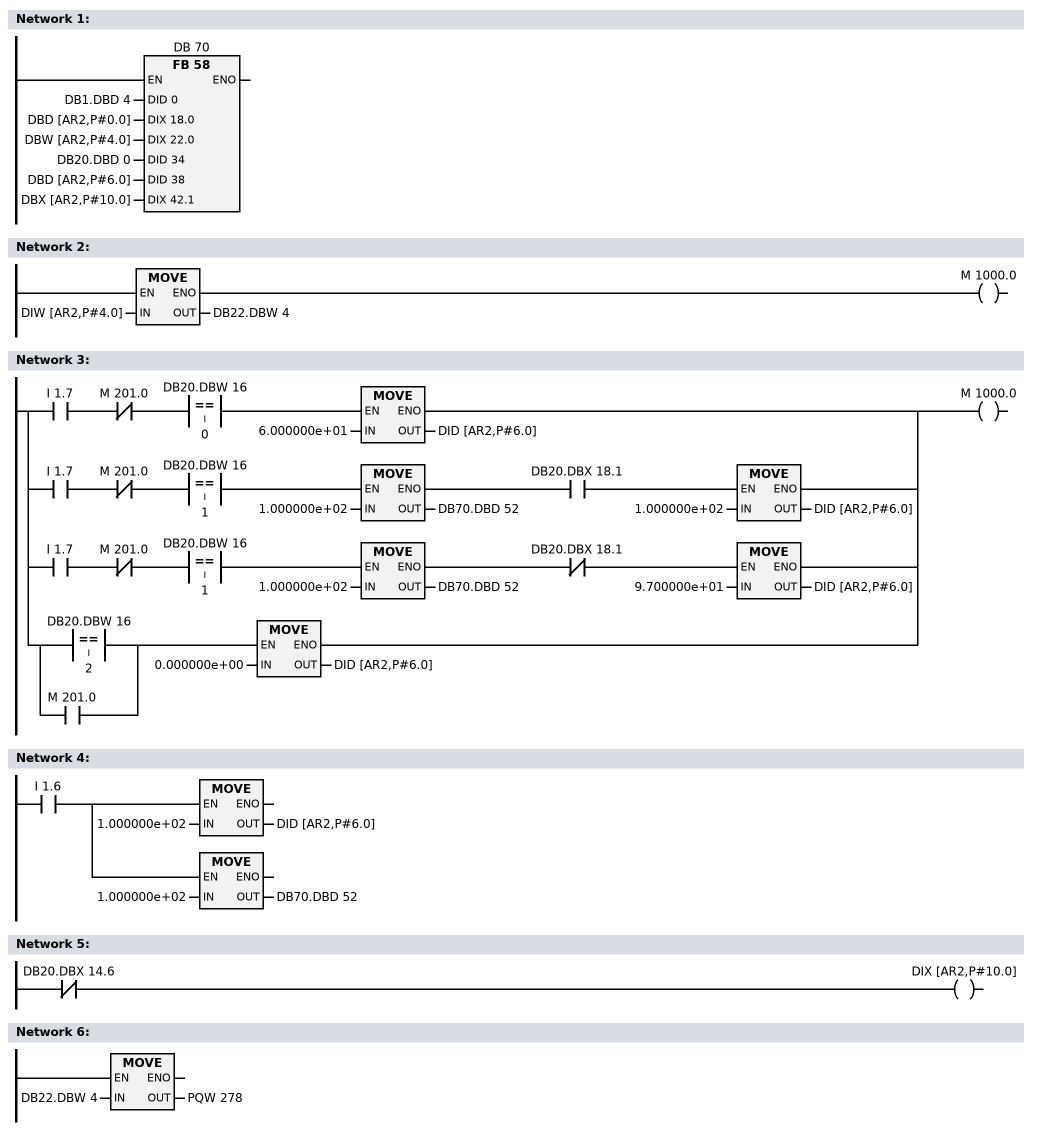
NETWORK
TITLE =
      CALL  FB 58 , DB 70 (
           DID 0                    := DB1.DBD 4,
           DIX 18.0                 := DBD [AR2,P#0.0],
           DIX 22.0                 := DBW [AR2,P#4.0],
           DID 34                   := DB20.DBD 0,
           DID 38                   := DBD [AR2,P#6.0],
           DIX 42.1                 := DBX [AR2,P#10.0]);
      NOP   0;
NETWORK
TITLE =
      L     DIW [AR2,P#4.0];
      T     DB22.DBW 4;
      SET;
      SAVE;
      CLR;
      A     BR;
      =     M 1000.0;
NETWORK
TITLE =
      O(;
      A     I 1.7;
      AN    M 201.0;
      A(;
      L     DB20.DBW 16;
      L     0;
      ==I;
      );
      JNB   M001;
      L     6.000000e+01;
      T     DID [AR2,P#6.0];
      SET;
      SAVE;
      CLR;
M001: A     BR;
      );
      O(;
      A(;
      A     I 1.7;
      AN    M 201.0;
      A(;
      L     DB20.DBW 16;
      L     1;
      ==I;
      );
      JNB   M002;
      L     1.000000e+02;
      T     DB70.DBD 52;
      SET;
      SAVE;
      CLR;
M002: A     BR;
      );
      A     DB20.DBX 18.1;
      JNB   M003;
      L     1.000000e+02;
      T     DID [AR2,P#6.0];
      SET;
      SAVE;
      CLR;
M003: A     BR;
      );
      O(;
      A(;
      A     I 1.7;
      AN    M 201.0;
      A(;
      L     DB20.DBW 16;
      L     1;
      ==I;
      );
      JNB   M004;
      L     1.000000e+02;
      T     DB70.DBD 52;
      SET;
      SAVE;
      CLR;
M004: A     BR;
      );
      AN    DB20.DBX 18.1;
      JNB   M005;
      L     9.700000e+01;
      T     DID [AR2,P#6.0];
      SET;
      SAVE;
      CLR;
M005: A     BR;
      );
      O(;
      A(;
      O(;
      L     DB20.DBW 16;
      L     2;
      ==I;
      );
      O     M 201.0;
      );
      JNB   M006;
      L     0.000000e+00;
      T     DID [AR2,P#6.0];
      SET;
      SAVE;
      CLR;
M006: A     BR;
      );
      =     M 1000.0;
NETWORK
TITLE =
      A     I 1.6;
      =     L 0.0;
      A     L 0.0;
      JNB   M007;
      L     1.000000e+02;
      T     DID [AR2,P#6.0];
M007: NOP   0;
      A     L 0.0;
      JNB   M008;
      L     1.000000e+02;
      T     DB70.DBD 52;
M008: NOP   0;
NETWORK
TITLE =
      AN    DB20.DBX 14.6;
      =     DIX [AR2,P#10.0];
NETWORK
TITLE =
      L     DB22.DBW 4;
      T     PQW 278;
      NOP   0;
END_FUNCTION_BLOCK

// FB 58: know-how protected block, not included

FUNCTION_BLOCK FB 94
VERSION : 0.1
BEGIN
// (block stored without names or comments; labels and parameter names are numbered)
NETWORK
TITLE =
      CALL  FB 20 , DB 120 (
           DIX 0.0                  := I 0.0,
           DIX 0.1                  := I 0.1,
           DIX 0.2                  := I 0.2,
           DIX 0.3                  := I 0.3,
           DIX 0.4                  := I 0.4,
           DIX 0.7                  := DB17.DBX 2.0,
           DIX 1.0                  := DB17.DBX 2.1,
           DIW 2                    := DB17.DBW 4,
           DIW 4                    := DB17.DBW 6,
           DID 6                    := DB17.DBD 8,
           DID 10                   := DB17.DBD 12,
           DIW 14                   := 10,
           DIW 16                   := 11,
           DIW 18                   := 12,
           DIW 20                   := 13,
           DIW 22                   := 14,
           DID 24                   := L#1092616192,
           DID 28                   := L#0,
           DID 32                   := L#1128792064,
           DID 36                   := L#0,
           DIW 40                   := DB17.DBW 38,
           DIX 42.0                 := DB17.DBX 40.1,
           DIX 42.1                 := DB17.DBX 40.2,
           DIX 46.1                 := DB2.DBX 16.0,
           DIW 52                   := 51,
           DIW 54                   := 52,
           DIW 56                   := 58,
           DIW 58                   := 61,
           DIX 60.0                 := Q 0.0,
           DIX 60.1                 := Q 0.1,
           DIX 60.2                 := Q 0.2,
           DIX 60.3                 := Q 0.3,
           DIX 60.4                 := DB17.DBX 16.0,
           DID 62                   := DB17.DBD 18,
           DIX 66.0                 := DB17.DBX 22.0,
           DIW 68                   := DB17.DBW 24,
           DID 70                   := DB17.DBD 26,
           DIX 74.0                 := Q 0.5,
           DIX 74.1                 := DB17.DBX 30.0,
           DIW 76                   := DB17.DBW 32,
           DID 78                   := DB17.DBD 34,
           DIX 82.0                 := Q 0.4,
           DIX 82.1                 := M 300.0,
           DIX 82.2                 := DB17.DBX 40.0,
           DIX 82.3                 := DB17.DBX 40.3,
           DIW 84                   := DB17.DBW 0);
NETWORK
TITLE =
      A     DB18.DBX 30.0;
      =     DB17.DBX 2.1;
      L     PIW 272;
      T     DB17.DBW 6;
      L     PIW 274;
      T     DB17.DBW 38;
      L     DB18.DBD 26;
      T     DB17.DBD 12;
      O     DB19.DBX 18.2;
      O     DB20.DBX 18.2;
      =     DB17.DBX 2.0;
      A     DB18.DBX 40.0;
      =     DB17.DBX 40.1;
      A     DB18.DBX 22.0;
      =     DB17.DBX 40.2;
END_FUNCTION_BLOCK

FUNCTION_BLOCK FB 95
VERSION : 0.1
BEGIN
// (block stored without names or comments; labels and parameter names are numbered)
NETWORK
TITLE =
      CALL  FB 20 , DB 230 (
           DIX 0.0                  := I 0.5,
           DIX 0.1                  := I 0.6,
           DIX 0.2                  := I 0.7,
           DIX 0.3                  := I 1.0,
           DIX 0.4                  := I 1.1,
           DIX 0.7                  := DB18.DBX 2.0,
           DIX 1.0                  := DB18.DBX 2.1,
           DIW 2                    := DB18.DBW 4,
           DIW 4                    := DB18.DBW 6,
           DID 6                    := DB18.DBD 8,
           DID 10                   := DB18.DBD 12,
           DIW 14                   := 20,
           DIW 16                   := 21,
           DIW 18                   := 22,
           DIW 20                   := 23,
           DIW 22                   := 24,
           DID 24                   := L#1092616192,
           DID 28                   := L#0,
           DID 32                   := L#1128792064,
           DID 36                   := L#0,
           DIW 40                   := DB18.DBW 38,
           DIX 42.0                 := DB18.DBX 40.1,
           DIX 42.1                 := DB18.DBX 40.2,
           DIX 46.1                 := DB2.DBX 16.0,
           DIW 52                   := 50,
           DIW 54                   := 53,
           DIW 56                   := 60,
           DIW 58                   := 62,
           DIX 60.0                 := Q 0.6,
           DIX 60.1                 := Q 0.7,
           DIX 60.2                 := Q 1.0,
           DIX 60.3                 := Q 1.1,
           DIX 60.4                 := DB18.DBX 16.0,
           DID 62                   := DB18.DBD 18,
           DIX 66.0                 := DB18.DBX 22.0,
           DIW 68                   := DB18.DBW 24,
           DID 70                   := DB18.DBD 26,
           DIX 74.0                 := Q 1.3,
           DIX 74.1                 := DB18.DBX 30.0,
           DIW 76                   := DB18.DBW 32,
           DID 78                   := DB18.DBD 34,
           DIX 82.0                 := Q 1.2,
           DIX 82.1                 := M 300.1,
           DIX 82.2                 := DB18.DBX 40.0,
           DIX 82.3                 := DB18.DBX 40.3,
           DIW 84                   := DB18.DBW 0);
NETWORK
TITLE =
      A     DB17.DBX 30.0;
      =     DB18.DBX 2.1;
      L     PIW 276;
      T     DB18.DBW 6;
      L     PIW 278;
      T     DB18.DBW 38;
      L     DB17.DBD 26;
      T     DB18.DBD 12;
      O     DB19.DBX 18.2;
      O     DB20.DBX 18.2;
      =     DB18.DBX 2.0;
      A     DB17.DBX 40.0;
      =     DB18.DBX 40.1;
      A     DB17.DBX 22.0;
      =     DB18.DBX 40.2;
END_FUNCTION_BLOCK

FUNCTION_BLOCK FB 98
VERSION : 0.1
BEGIN
// (block stored without names or comments; labels and parameter names are numbered)
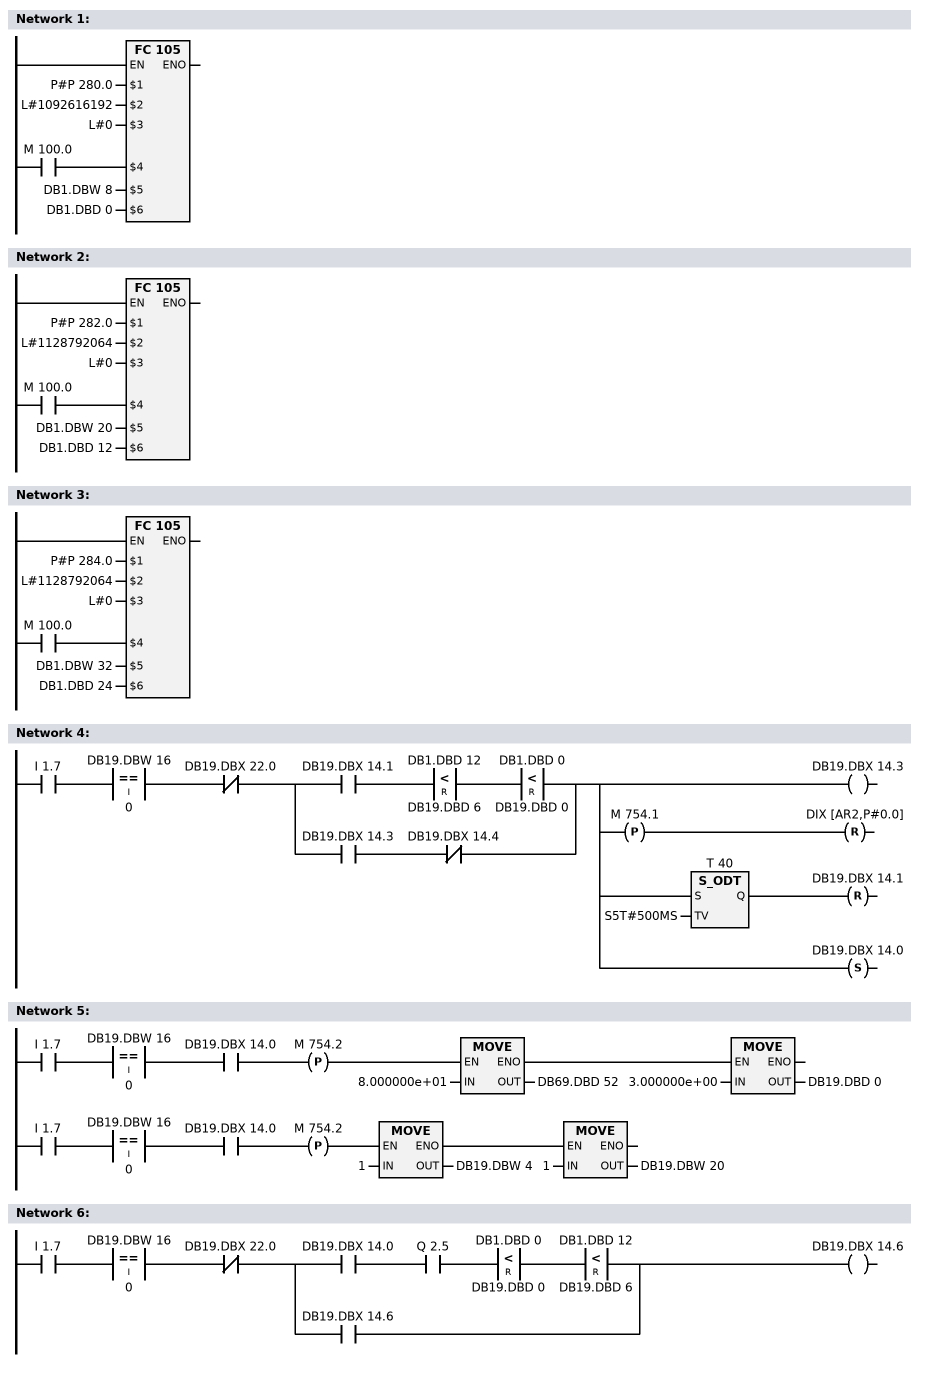
NETWORK
TITLE =
      A     M 100.0;
      =     L 2.0;
      BLD   103;
      CALL  FC 105 (
           $1                       := P#P 280.0,
           $2                       := L#1092616192,
           $3                       := L#0,
           $4                       := L 2.0,
           $5                       := DB1.DBW 8,
           $6                       := DB1.DBD 0);
      NOP   0;
NETWORK
TITLE =
      A     M 100.0;
      =     L 2.0;
      BLD   103;
      CALL  FC 105 (
           $1                       := P#P 282.0,
           $2                       := L#1128792064,
           $3                       := L#0,
           $4                       := L 2.0,
           $5                       := DB1.DBW 20,
           $6                       := DB1.DBD 12);
      NOP   0;
NETWORK
TITLE =
      A     M 100.0;
      =     L 2.0;
      BLD   103;
      CALL  FC 105 (
           $1                       := P#P 284.0,
           $2                       := L#1128792064,
           $3                       := L#0,
           $4                       := L 2.0,
           $5                       := DB1.DBW 32,
           $6                       := DB1.DBD 24);
      NOP   0;
NETWORK
TITLE =
      A     I 1.7;
      A(;
      L     DB19.DBW 16;
      L     0;
      ==I;
      );
      AN    DB19.DBX 22.0;
      A(;
      A     DB19.DBX 14.1;
      A(;
      L     DB1.DBD 12;
      L     DB19.DBD 6;
      <R;
      );
      A(;
      L     DB1.DBD 0;
      L     DB19.DBD 0;
      <R;
      );
      O;
      A     DB19.DBX 14.3;
      AN    DB19.DBX 14.4;
      );
      =     L 2.0;
      A     L 2.0;
      BLD   102;
      =     DB19.DBX 14.3;
      A     L 2.0;
      FP    M 754.1;
      R     DIX [AR2,P#0.0];
      A     L 2.0;
      L     S5T#500MS;
      SD    T 40;
      NOP   0;
      NOP   0;
      NOP   0;
      A     T 40;
      R     DB19.DBX 14.1;
      A     L 2.0;
      BLD   102;
      S     DB19.DBX 14.0;
NETWORK
TITLE =
      A     I 1.7;
      A(;
      L     DB19.DBW 16;
      L     0;
      ==I;
      );
      A     DB19.DBX 14.0;
      FP    M 754.2;
      =     L 2.0;
      A(;
      A     L 2.0;
      JNB   M001;
      L     8.000000e+01;
      T     DB69.DBD 52;
      SET;
      SAVE;
      CLR;
M001: A     BR;
      );
      JNB   M002;
      L     3.000000e+00;
      T     DB19.DBD 0;
M002: NOP   0;
      A(;
      A     L 2.0;
      JNB   M003;
      L     1;
      T     DB19.DBW 4;
      SET;
      SAVE;
      CLR;
M003: A     BR;
      );
      JNB   M004;
      L     1;
      T     DB19.DBW 20;
M004: NOP   0;
NETWORK
TITLE =
      A     I 1.7;
      A(;
      L     DB19.DBW 16;
      L     0;
      ==I;
      );
      AN    DB19.DBX 22.0;
      A(;
      A     DB19.DBX 14.0;
      A     Q 2.5;
      A(;
      L     DB1.DBD 0;
      L     DB19.DBD 0;
      <R;
      );
      A(;
      L     DB1.DBD 12;
      L     DB19.DBD 6;
      <R;
      );
      O     DB19.DBX 14.6;
      );
      =     DB19.DBX 14.6;
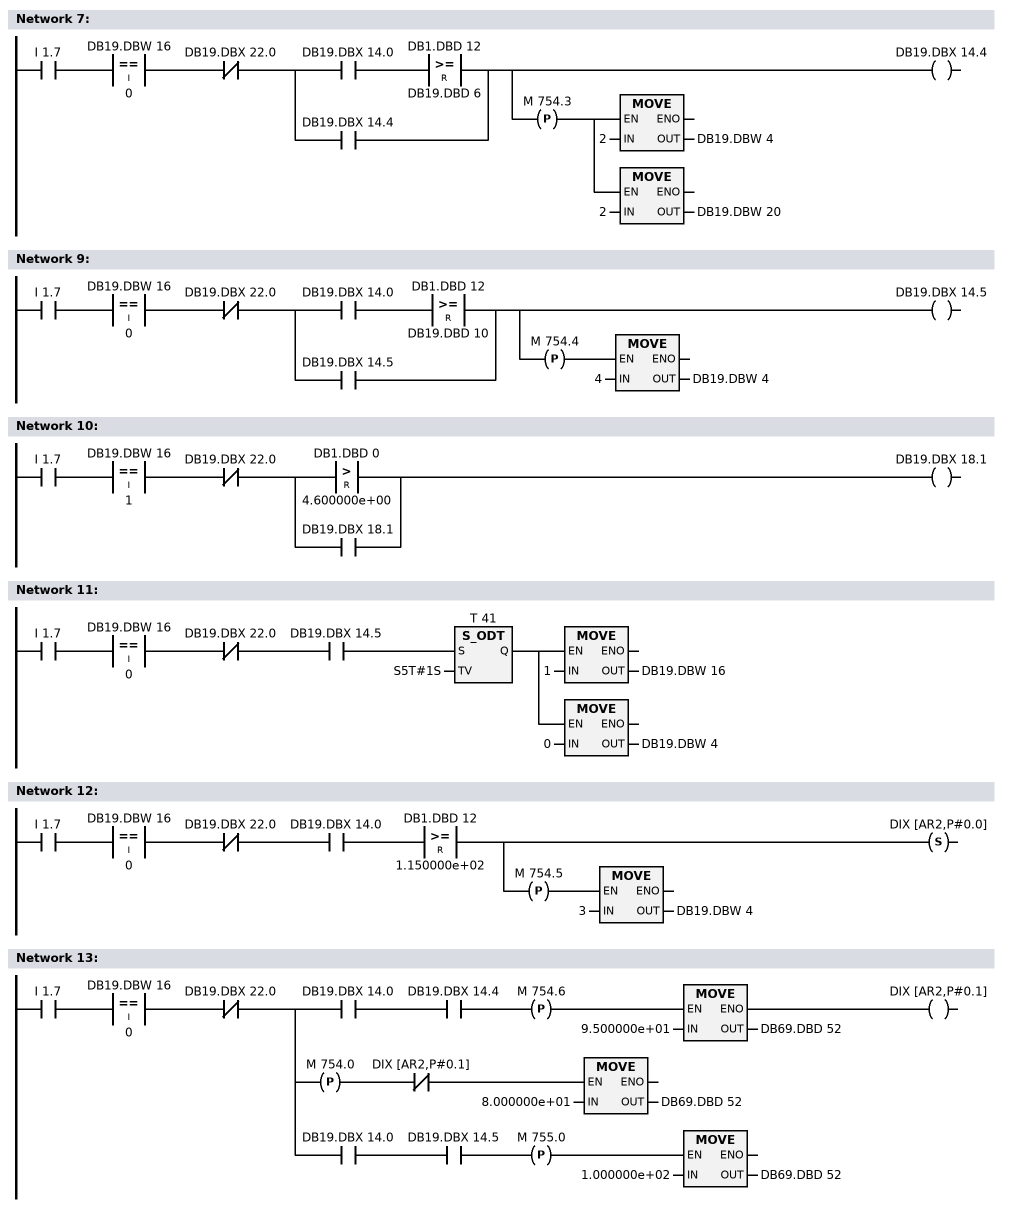
NETWORK
TITLE =
      A     I 1.7;
      A(;
      L     DB19.DBW 16;
      L     0;
      ==I;
      );
      AN    DB19.DBX 22.0;
      A(;
      A     DB19.DBX 14.0;
      A(;
      L     DB1.DBD 12;
      L     DB19.DBD 6;
      >=R;
      );
      O     DB19.DBX 14.4;
      );
      =     L 2.0;
      A     L 2.0;
      BLD   102;
      =     DB19.DBX 14.4;
      A     L 2.0;
      FP    M 754.3;
      =     L 2.1;
      A     L 2.1;
      JNB   M005;
      L     2;
      T     DB19.DBW 4;
M005: NOP   0;
      A     L 2.1;
      JNB   M006;
      L     2;
      T     DB19.DBW 20;
M006: NOP   0;
NETWORK
TITLE =
      A(;
      A     DB19.DBX 14.4;
      FP    M 101.1;
      S     M 101.0;
      A(;
      O(;
      L     DB19.DBW 16;
      L     1;
      ==I;
      );
      O     DB19.DBX 22.0;
      );
      R     M 101.0;
      A     M 101.0;
      );
      L     S5T#1M30S;
      SD    T 57;
      NOP   0;
      NOP   0;
      NOP   0;
      A     T 57;
      =     DB19.DBX 38.0;
NETWORK
TITLE =
      A     I 1.7;
      A(;
      L     DB19.DBW 16;
      L     0;
      ==I;
      );
      AN    DB19.DBX 22.0;
      A(;
      A     DB19.DBX 14.0;
      A(;
      L     DB1.DBD 12;
      L     DB19.DBD 10;
      >=R;
      );
      O     DB19.DBX 14.5;
      );
      =     L 2.0;
      A     L 2.0;
      BLD   102;
      =     DB19.DBX 14.5;
      A     L 2.0;
      FP    M 754.4;
      JNB   M007;
      L     4;
      T     DB19.DBW 4;
M007: NOP   0;
NETWORK
TITLE =
      A     I 1.7;
      A(;
      L     DB19.DBW 16;
      L     1;
      ==I;
      );
      AN    DB19.DBX 22.0;
      A(;
      O(;
      L     DB1.DBD 0;
      L     4.600000e+00;
      >R;
      );
      O     DB19.DBX 18.1;
      );
      =     DB19.DBX 18.1;
NETWORK
TITLE =
      A     I 1.7;
      A(;
      L     DB19.DBW 16;
      L     0;
      ==I;
      );
      AN    DB19.DBX 22.0;
      A     DB19.DBX 14.5;
      L     S5T#1S;
      SD    T 41;
      NOP   0;
      NOP   0;
      NOP   0;
      A     T 41;
      =     L 2.0;
      A     L 2.0;
      JNB   M008;
      L     1;
      T     DB19.DBW 16;
M008: NOP   0;
      A     L 2.0;
      JNB   M009;
      L     0;
      T     DB19.DBW 4;
M009: NOP   0;
NETWORK
TITLE =
      A     I 1.7;
      A(;
      L     DB19.DBW 16;
      L     0;
      ==I;
      );
      AN    DB19.DBX 22.0;
      A     DB19.DBX 14.0;
      A(;
      L     DB1.DBD 12;
      L     1.150000e+02;
      >=R;
      );
      =     L 2.0;
      A     L 2.0;
      BLD   102;
      S     DIX [AR2,P#0.0];
      A     L 2.0;
      FP    M 754.5;
      JNB   M010;
      L     3;
      T     DB19.DBW 4;
M010: NOP   0;
NETWORK
TITLE =
      A     I 1.7;
      A(;
      L     DB19.DBW 16;
      L     0;
      ==I;
      );
      AN    DB19.DBX 22.0;
      =     L 2.0;
      A     L 2.0;
      A     DB19.DBX 14.0;
      A     DB19.DBX 14.4;
      FP    M 754.6;
      JNB   M011;
      L     9.500000e+01;
      T     DB69.DBD 52;
      SET;
      SAVE;
      CLR;
M011: A     BR;
      =     DIX [AR2,P#0.1];
      A     L 2.0;
      FP    M 754.0;
      AN    DIX [AR2,P#0.1];
      JNB   M012;
      L     8.000000e+01;
      T     DB69.DBD 52;
M012: NOP   0;
      A     L 2.0;
      A     DB19.DBX 14.0;
      A     DB19.DBX 14.5;
      FP    M 755.0;
      JNB   M013;
      L     1.000000e+02;
      T     DB69.DBD 52;
M013: NOP   0;
NETWORK
TITLE =
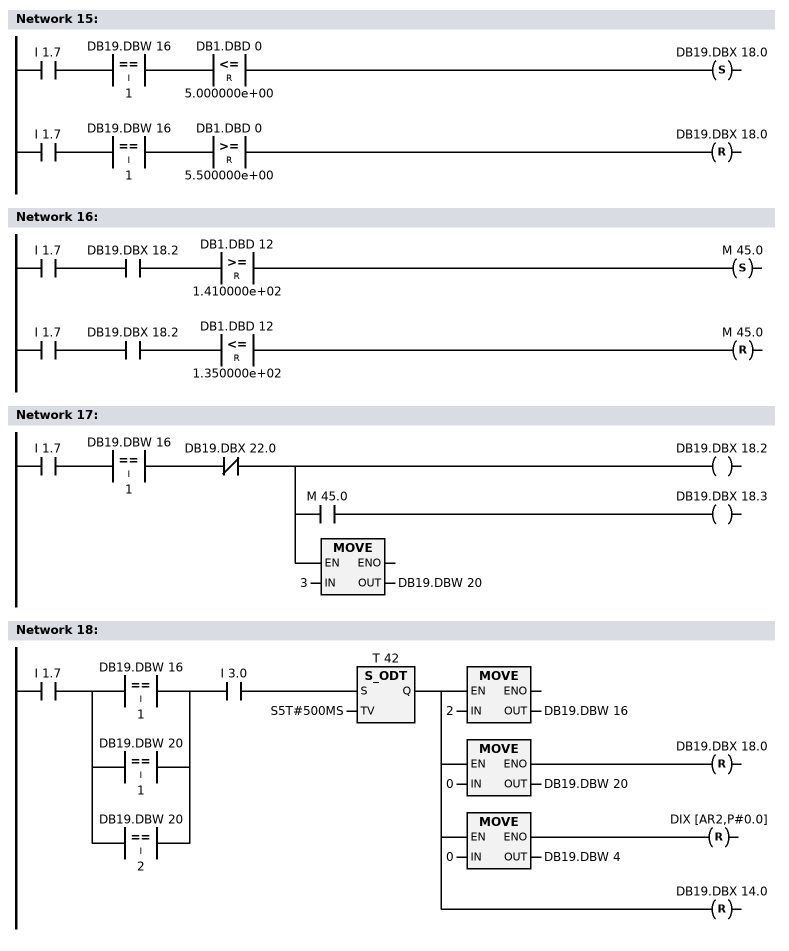
NETWORK
TITLE =
      A     I 1.7;
      A(;
      L     DB19.DBW 16;
      L     1;
      ==I;
      );
      A(;
      L     DB1.DBD 0;
      L     5.000000e+00;
      <=R;
      );
      S     DB19.DBX 18.0;
      A     I 1.7;
      A(;
      L     DB19.DBW 16;
      L     1;
      ==I;
      );
      A(;
      L     DB1.DBD 0;
      L     5.500000e+00;
      >=R;
      );
      R     DB19.DBX 18.0;
      NOP   0;
NETWORK
TITLE =
      A     I 1.7;
      A     DB19.DBX 18.2;
      A(;
      L     DB1.DBD 12;
      L     1.410000e+02;
      >=R;
      );
      S     M 45.0;
      A     I 1.7;
      A     DB19.DBX 18.2;
      A(;
      L     DB1.DBD 12;
      L     1.350000e+02;
      <=R;
      );
      R     M 45.0;
      NOP   0;
NETWORK
TITLE =
      A     I 1.7;
      A(;
      L     DB19.DBW 16;
      L     1;
      ==I;
      );
      AN    DB19.DBX 22.0;
      =     L 2.0;
      A     L 2.0;
      BLD   102;
      =     DB19.DBX 18.2;
      A     L 2.0;
      A     M 45.0;
      =     DB19.DBX 18.3;
      A     L 2.0;
      JNB   M014;
      L     3;
      T     DB19.DBW 20;
M014: NOP   0;
NETWORK
TITLE =
      A     I 1.7;
      A(;
      O(;
      L     DB19.DBW 16;
      L     1;
      ==I;
      );
      O(;
      L     DB19.DBW 20;
      L     1;
      ==I;
      );
      O(;
      L     DB19.DBW 20;
      L     2;
      ==I;
      );
      );
      A     I 3.0;
      L     S5T#500MS;
      SD    T 42;
      NOP   0;
      NOP   0;
      NOP   0;
      A     T 42;
      =     L 2.0;
      A     L 2.0;
      JNB   M015;
      L     2;
      T     DB19.DBW 16;
M015: NOP   0;
      A     L 2.0;
      JNB   M016;
      L     0;
      T     DB19.DBW 20;
      SET;
      SAVE;
      CLR;
M016: A     BR;
      R     DB19.DBX 18.0;
      A     L 2.0;
      JNB   M017;
      L     0;
      T     DB19.DBW 4;
      SET;
      SAVE;
      CLR;
M017: A     BR;
      R     DIX [AR2,P#0.0];
      A     L 2.0;
      BLD   102;
      R     DB19.DBX 14.0;
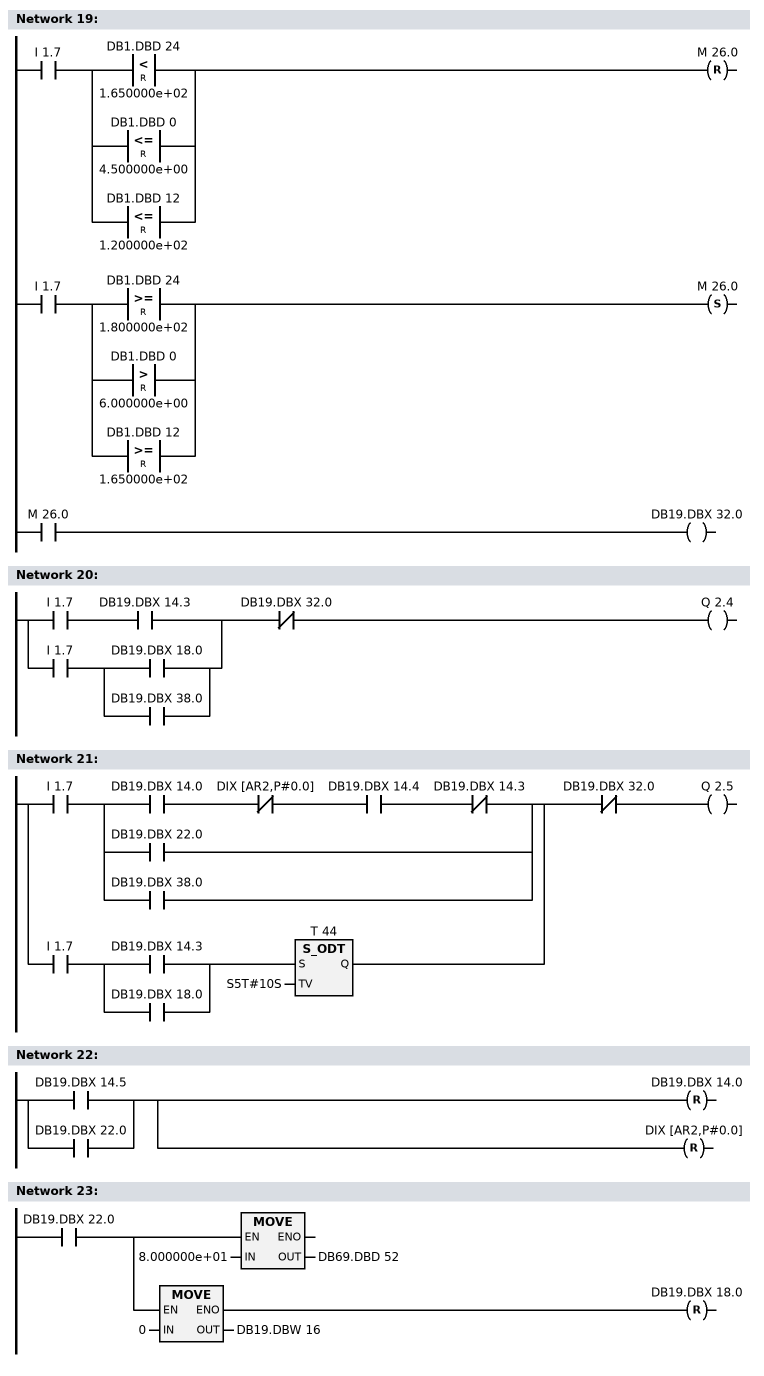
NETWORK
TITLE =
      A     I 1.7;
      A(;
      O(;
      L     DB1.DBD 24;
      L     1.650000e+02;
      <R;
      );
      O(;
      L     DB1.DBD 0;
      L     4.500000e+00;
      <=R;
      );
      O(;
      L     DB1.DBD 12;
      L     1.200000e+02;
      <=R;
      );
      );
      R     M 26.0;
      A     I 1.7;
      A(;
      O(;
      L     DB1.DBD 24;
      L     1.800000e+02;
      >=R;
      );
      O(;
      L     DB1.DBD 0;
      L     6.000000e+00;
      >R;
      );
      O(;
      L     DB1.DBD 12;
      L     1.650000e+02;
      >=R;
      );
      );
      S     M 26.0;
      A     M 26.0;
      =     DB19.DBX 32.0;
NETWORK
TITLE =
      A(;
      A     I 1.7;
      A     DB19.DBX 14.3;
      O;
      A     I 1.7;
      A(;
      O     DB19.DBX 18.0;
      O     DB19.DBX 38.0;
      );
      );
      AN    DB19.DBX 32.0;
      =     Q 2.4;
NETWORK
TITLE =
      A(;
      A     I 1.7;
      A(;
      A     DB19.DBX 14.0;
      AN    DIX [AR2,P#0.0];
      A     DB19.DBX 14.4;
      AN    DB19.DBX 14.3;
      O     DB19.DBX 22.0;
      O     DB19.DBX 38.0;
      );
      O(;
      A     I 1.7;
      A(;
      O     DB19.DBX 14.3;
      O     DB19.DBX 18.0;
      );
      L     S5T#10S;
      SD    T 44;
      NOP   0;
      NOP   0;
      NOP   0;
      A     T 44;
      );
      );
      AN    DB19.DBX 32.0;
      =     Q 2.5;
NETWORK
TITLE =
      O     DB19.DBX 14.5;
      O     DB19.DBX 22.0;
      R     DB19.DBX 14.0;
      R     DIX [AR2,P#0.0];
NETWORK
TITLE =
      A     DB19.DBX 22.0;
      =     L 2.0;
      A     L 2.0;
      JNB   M018;
      L     8.000000e+01;
      T     DB69.DBD 52;
M018: NOP   0;
      A     L 2.0;
      JNB   M019;
      L     0;
      T     DB19.DBW 16;
      SET;
      SAVE;
      CLR;
M019: A     BR;
      R     DB19.DBX 18.0;
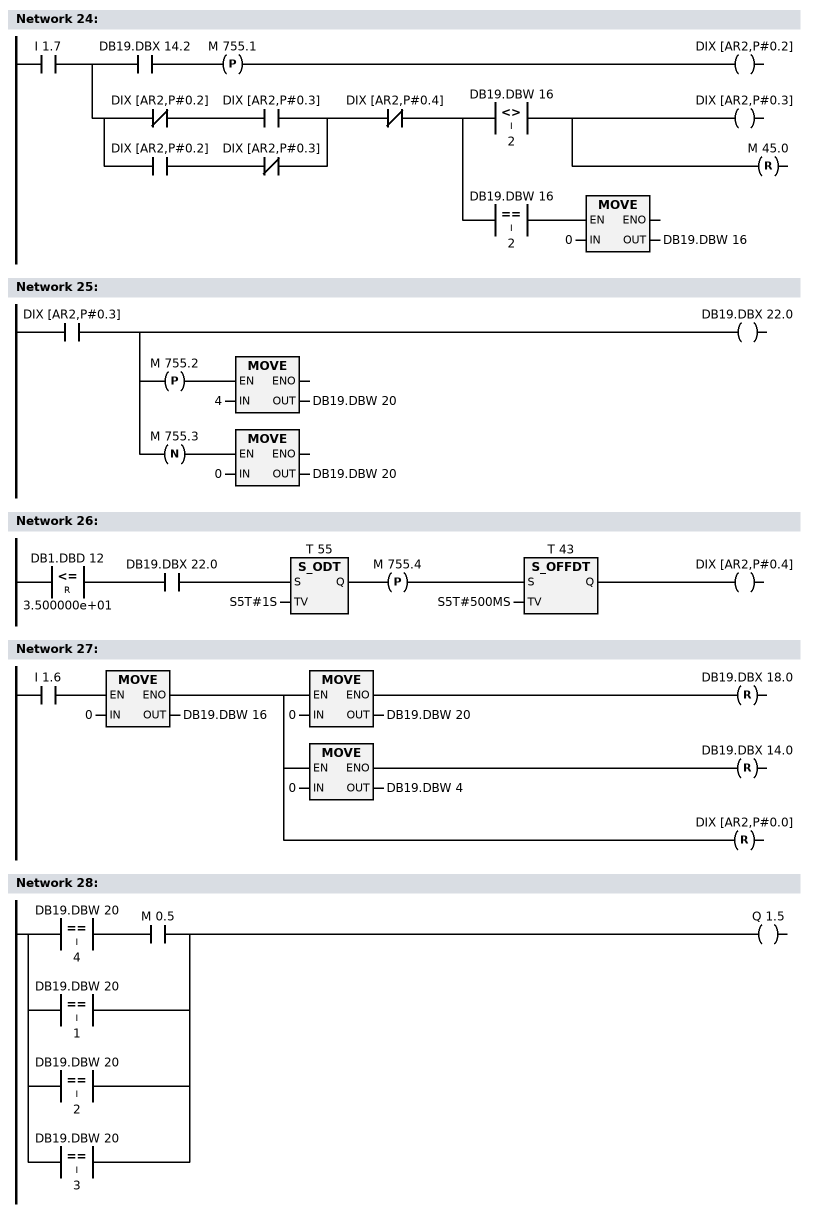
NETWORK
TITLE =
      A     I 1.7;
      =     L 2.0;
      A     L 2.0;
      A     DB19.DBX 14.2;
      FP    M 755.1;
      =     DIX [AR2,P#0.2];
      A     L 2.0;
      A(;
      AN    DIX [AR2,P#0.2];
      A     DIX [AR2,P#0.3];
      O;
      A     DIX [AR2,P#0.2];
      AN    DIX [AR2,P#0.3];
      );
      AN    DIX [AR2,P#0.4];
      =     L 2.1;
      A     L 2.1;
      A(;
      L     DB19.DBW 16;
      L     2;
      <>I;
      );
      =     DIX [AR2,P#0.3];
      R     M 45.0;
      A     L 2.1;
      A(;
      L     DB19.DBW 16;
      L     2;
      ==I;
      );
      JNB   M020;
      L     0;
      T     DB19.DBW 16;
M020: NOP   0;
NETWORK
TITLE =
      A     DIX [AR2,P#0.3];
      =     L 2.0;
      A     L 2.0;
      BLD   102;
      =     DB19.DBX 22.0;
      A     L 2.0;
      FP    M 755.2;
      JNB   M021;
      L     4;
      T     DB19.DBW 20;
M021: NOP   0;
      A     L 2.0;
      FN    M 755.3;
      JNB   M022;
      L     0;
      T     DB19.DBW 20;
M022: NOP   0;
NETWORK
TITLE =
      A(;
      A(;
      L     DB1.DBD 12;
      L     3.500000e+01;
      <=R;
      );
      A     DB19.DBX 22.0;
      L     S5T#1S;
      SD    T 55;
      NOP   0;
      NOP   0;
      NOP   0;
      A     T 55;
      );
      FP    M 755.4;
      L     S5T#500MS;
      SF    T 43;
      NOP   0;
      NOP   0;
      NOP   0;
      A     T 43;
      =     DIX [AR2,P#0.4];
NETWORK
TITLE =
      A     I 1.6;
      JNB   M023;
      L     0;
      T     DB19.DBW 16;
      SET;
      SAVE;
      CLR;
M023: A     BR;
      =     L 2.0;
      A     L 2.0;
      JNB   M024;
      L     0;
      T     DB19.DBW 20;
      SET;
      SAVE;
      CLR;
M024: A     BR;
      R     DB19.DBX 18.0;
      A     L 2.0;
      JNB   M025;
      L     0;
      T     DB19.DBW 4;
      SET;
      SAVE;
      CLR;
M025: A     BR;
      R     DB19.DBX 14.0;
      A     L 2.0;
      BLD   102;
      R     DIX [AR2,P#0.0];
NETWORK
TITLE =
      A(;
      L     DB19.DBW 20;
      L     4;
      ==I;
      );
      A     M 0.5;
      O(;
      L     DB19.DBW 20;
      L     1;
      ==I;
      );
      O(;
      L     DB19.DBW 20;
      L     2;
      ==I;
      );
      O(;
      L     DB19.DBW 20;
      L     3;
      ==I;
      );
      =     Q 1.5;
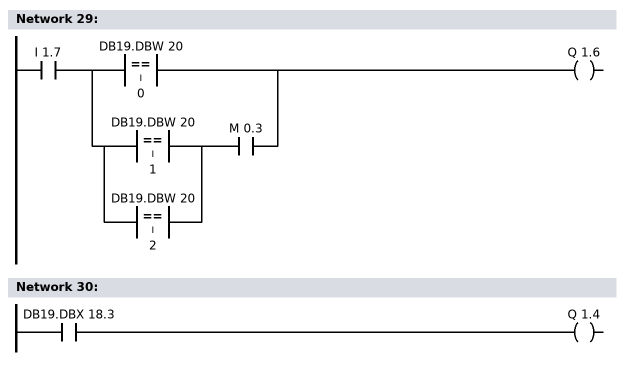
NETWORK
TITLE =
      A     I 1.7;
      A(;
      O(;
      L     DB19.DBW 20;
      L     0;
      ==I;
      );
      O;
      A(;
      O(;
      L     DB19.DBW 20;
      L     1;
      ==I;
      );
      O(;
      L     DB19.DBW 20;
      L     2;
      ==I;
      );
      );
      A     M 0.3;
      );
      =     Q 1.6;
NETWORK
TITLE =
      A     DB19.DBX 18.3;
      =     Q 1.4;
END_FUNCTION_BLOCK

FUNCTION_BLOCK FB 99
VERSION : 0.1
BEGIN
// (block stored without names or comments; labels and parameter names are numbered)
NETWORK
TITLE =
      A     M 100.0;
      =     L 0.0;
      BLD   103;
      A(;
      A     M 100.0;
      =     L 0.1;
      BLD   103;
      CALL  FC 105 (
           $1                       := P#P 286.0,
           $2                       := L#1092616192,
           $3                       := L#0,
           $4                       := L 0.1,
           $5                       := DB1.DBW 10,
           $6                       := DB1.DBD 4);
      A     BR;
      );
      JNB   M001;
      CALL  FC 105 (
           $1                       := P#P 288.0,
           $2                       := L#1128792064,
           $3                       := L#0,
           $4                       := L 0.0,
           $5                       := DB1.DBW 22,
           $6                       := DB1.DBD 16);
M001: NOP   0;
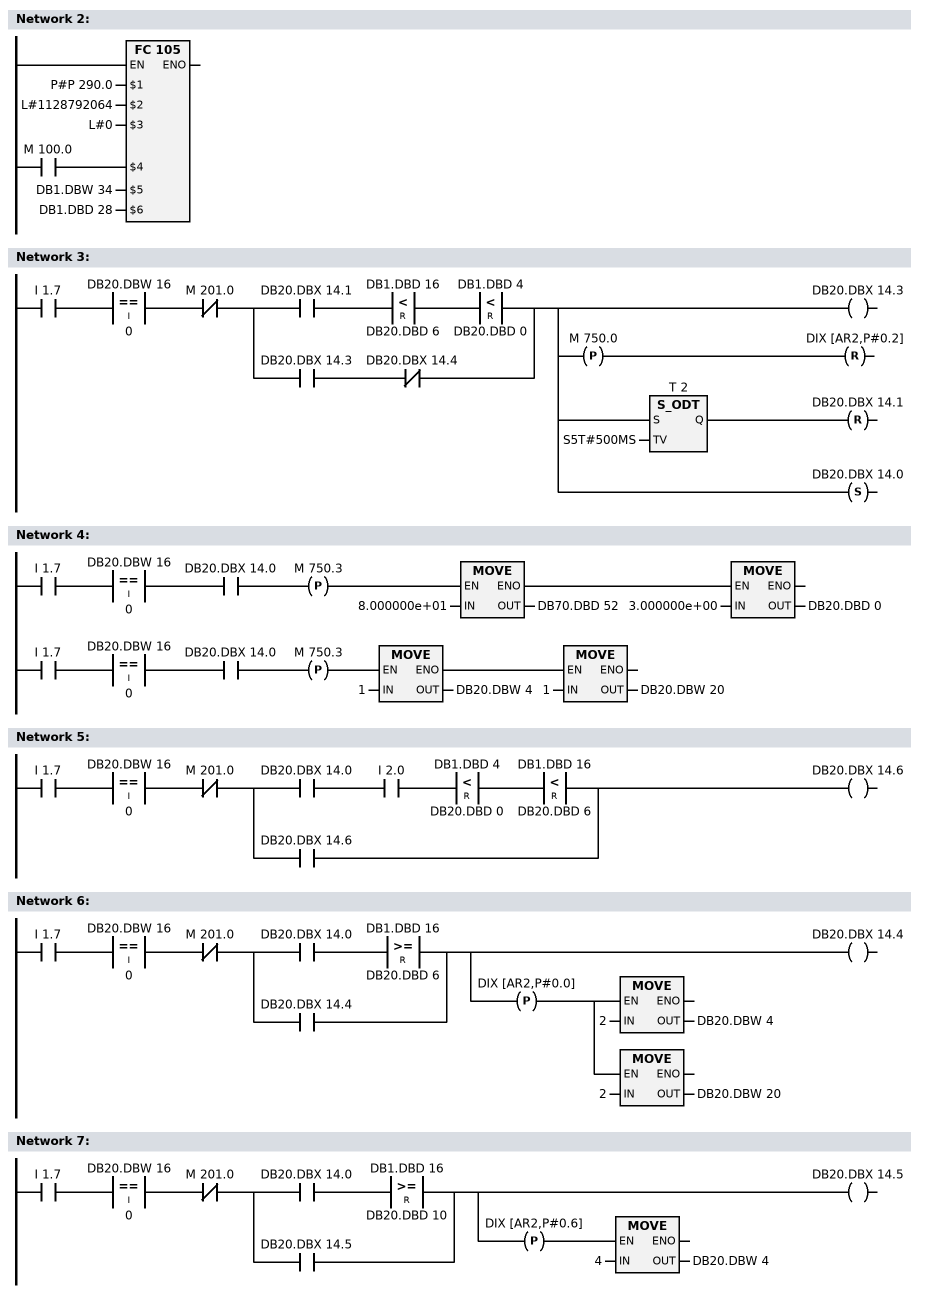
NETWORK
TITLE =
      A     M 100.0;
      =     L 0.0;
      BLD   103;
      CALL  FC 105 (
           $1                       := P#P 290.0,
           $2                       := L#1128792064,
           $3                       := L#0,
           $4                       := L 0.0,
           $5                       := DB1.DBW 34,
           $6                       := DB1.DBD 28);
      NOP   0;
NETWORK
TITLE =
      A     I 1.7;
      A(;
      L     DB20.DBW 16;
      L     0;
      ==I;
      );
      AN    M 201.0;
      A(;
      A     DB20.DBX 14.1;
      A(;
      L     DB1.DBD 16;
      L     DB20.DBD 6;
      <R;
      );
      A(;
      L     DB1.DBD 4;
      L     DB20.DBD 0;
      <R;
      );
      O;
      A     DB20.DBX 14.3;
      AN    DB20.DBX 14.4;
      );
      =     L 0.0;
      A     L 0.0;
      BLD   102;
      =     DB20.DBX 14.3;
      A     L 0.0;
      FP    M 750.0;
      R     DIX [AR2,P#0.2];
      A     L 0.0;
      L     S5T#500MS;
      SD    T 2;
      NOP   0;
      NOP   0;
      NOP   0;
      A     T 2;
      R     DB20.DBX 14.1;
      A     L 0.0;
      BLD   102;
      S     DB20.DBX 14.0;
NETWORK
TITLE =
      A     I 1.7;
      A(;
      L     DB20.DBW 16;
      L     0;
      ==I;
      );
      A     DB20.DBX 14.0;
      FP    M 750.3;
      =     L 0.0;
      A(;
      A     L 0.0;
      JNB   M002;
      L     8.000000e+01;
      T     DB70.DBD 52;
      SET;
      SAVE;
      CLR;
M002: A     BR;
      );
      JNB   M003;
      L     3.000000e+00;
      T     DB20.DBD 0;
M003: NOP   0;
      A(;
      A     L 0.0;
      JNB   M004;
      L     1;
      T     DB20.DBW 4;
      SET;
      SAVE;
      CLR;
M004: A     BR;
      );
      JNB   M005;
      L     1;
      T     DB20.DBW 20;
M005: NOP   0;
NETWORK
TITLE =
      A     I 1.7;
      A(;
      L     DB20.DBW 16;
      L     0;
      ==I;
      );
      AN    M 201.0;
      A(;
      A     DB20.DBX 14.0;
      A     I 2.0;
      A(;
      L     DB1.DBD 4;
      L     DB20.DBD 0;
      <R;
      );
      A(;
      L     DB1.DBD 16;
      L     DB20.DBD 6;
      <R;
      );
      O     DB20.DBX 14.6;
      );
      =     DB20.DBX 14.6;
NETWORK
TITLE =
      A     I 1.7;
      A(;
      L     DB20.DBW 16;
      L     0;
      ==I;
      );
      AN    M 201.0;
      A(;
      A     DB20.DBX 14.0;
      A(;
      L     DB1.DBD 16;
      L     DB20.DBD 6;
      >=R;
      );
      O     DB20.DBX 14.4;
      );
      =     L 0.0;
      A     L 0.0;
      BLD   102;
      =     DB20.DBX 14.4;
      A     L 0.0;
      FP    DIX [AR2,P#0.0];
      =     L 0.1;
      A     L 0.1;
      JNB   M006;
      L     2;
      T     DB20.DBW 4;
M006: NOP   0;
      A     L 0.1;
      JNB   M007;
      L     2;
      T     DB20.DBW 20;
M007: NOP   0;
NETWORK
TITLE =
      A     I 1.7;
      A(;
      L     DB20.DBW 16;
      L     0;
      ==I;
      );
      AN    M 201.0;
      A(;
      A     DB20.DBX 14.0;
      A(;
      L     DB1.DBD 16;
      L     DB20.DBD 10;
      >=R;
      );
      O     DB20.DBX 14.5;
      );
      =     L 0.0;
      A     L 0.0;
      BLD   102;
      =     DB20.DBX 14.5;
      A     L 0.0;
      FP    DIX [AR2,P#0.6];
      JNB   M008;
      L     4;
      T     DB20.DBW 4;
M008: NOP   0;
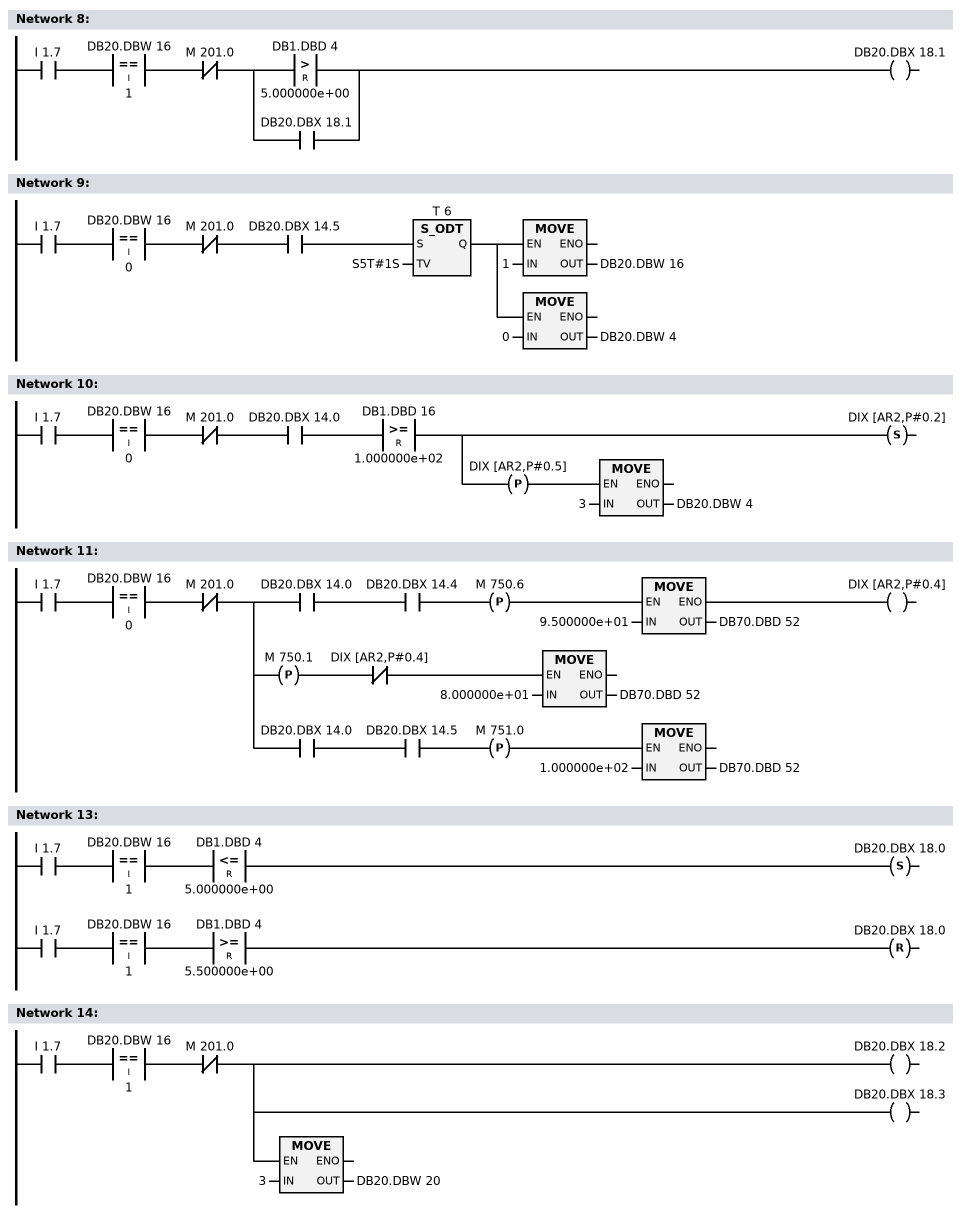
NETWORK
TITLE =
      A     I 1.7;
      A(;
      L     DB20.DBW 16;
      L     1;
      ==I;
      );
      AN    M 201.0;
      A(;
      O(;
      L     DB1.DBD 4;
      L     5.000000e+00;
      >R;
      );
      O     DB20.DBX 18.1;
      );
      =     DB20.DBX 18.1;
NETWORK
TITLE =
      A     I 1.7;
      A(;
      L     DB20.DBW 16;
      L     0;
      ==I;
      );
      AN    M 201.0;
      A     DB20.DBX 14.5;
      L     S5T#1S;
      SD    T 6;
      NOP   0;
      NOP   0;
      NOP   0;
      A     T 6;
      =     L 0.0;
      A     L 0.0;
      JNB   M009;
      L     1;
      T     DB20.DBW 16;
M009: NOP   0;
      A     L 0.0;
      JNB   M010;
      L     0;
      T     DB20.DBW 4;
M010: NOP   0;
NETWORK
TITLE =
      A     I 1.7;
      A(;
      L     DB20.DBW 16;
      L     0;
      ==I;
      );
      AN    M 201.0;
      A     DB20.DBX 14.0;
      A(;
      L     DB1.DBD 16;
      L     1.000000e+02;
      >=R;
      );
      =     L 0.0;
      A     L 0.0;
      BLD   102;
      S     DIX [AR2,P#0.2];
      A     L 0.0;
      FP    DIX [AR2,P#0.5];
      JNB   M011;
      L     3;
      T     DB20.DBW 4;
M011: NOP   0;
NETWORK
TITLE =
      A     I 1.7;
      A(;
      L     DB20.DBW 16;
      L     0;
      ==I;
      );
      AN    M 201.0;
      =     L 0.0;
      A     L 0.0;
      A     DB20.DBX 14.0;
      A     DB20.DBX 14.4;
      FP    M 750.6;
      JNB   M012;
      L     9.500000e+01;
      T     DB70.DBD 52;
      SET;
      SAVE;
      CLR;
M012: A     BR;
      =     DIX [AR2,P#0.4];
      A     L 0.0;
      FP    M 750.1;
      AN    DIX [AR2,P#0.4];
      JNB   M013;
      L     8.000000e+01;
      T     DB70.DBD 52;
M013: NOP   0;
      A     L 0.0;
      A     DB20.DBX 14.0;
      A     DB20.DBX 14.5;
      FP    M 751.0;
      JNB   M014;
      L     1.000000e+02;
      T     DB70.DBD 52;
M014: NOP   0;
NETWORK
TITLE =
NETWORK
TITLE =
      A     I 1.7;
      A(;
      L     DB20.DBW 16;
      L     1;
      ==I;
      );
      A(;
      L     DB1.DBD 4;
      L     5.000000e+00;
      <=R;
      );
      S     DB20.DBX 18.0;
      A     I 1.7;
      A(;
      L     DB20.DBW 16;
      L     1;
      ==I;
      );
      A(;
      L     DB1.DBD 4;
      L     5.500000e+00;
      >=R;
      );
      R     DB20.DBX 18.0;
      NOP   0;
NETWORK
TITLE =
      A     I 1.7;
      A(;
      L     DB20.DBW 16;
      L     1;
      ==I;
      );
      AN    M 201.0;
      =     L 0.0;
      A     L 0.0;
      BLD   102;
      =     DB20.DBX 18.2;
      A     L 0.0;
      BLD   102;
      =     DB20.DBX 18.3;
      A     L 0.0;
      JNB   M015;
      L     3;
      T     DB20.DBW 20;
M015: NOP   0;
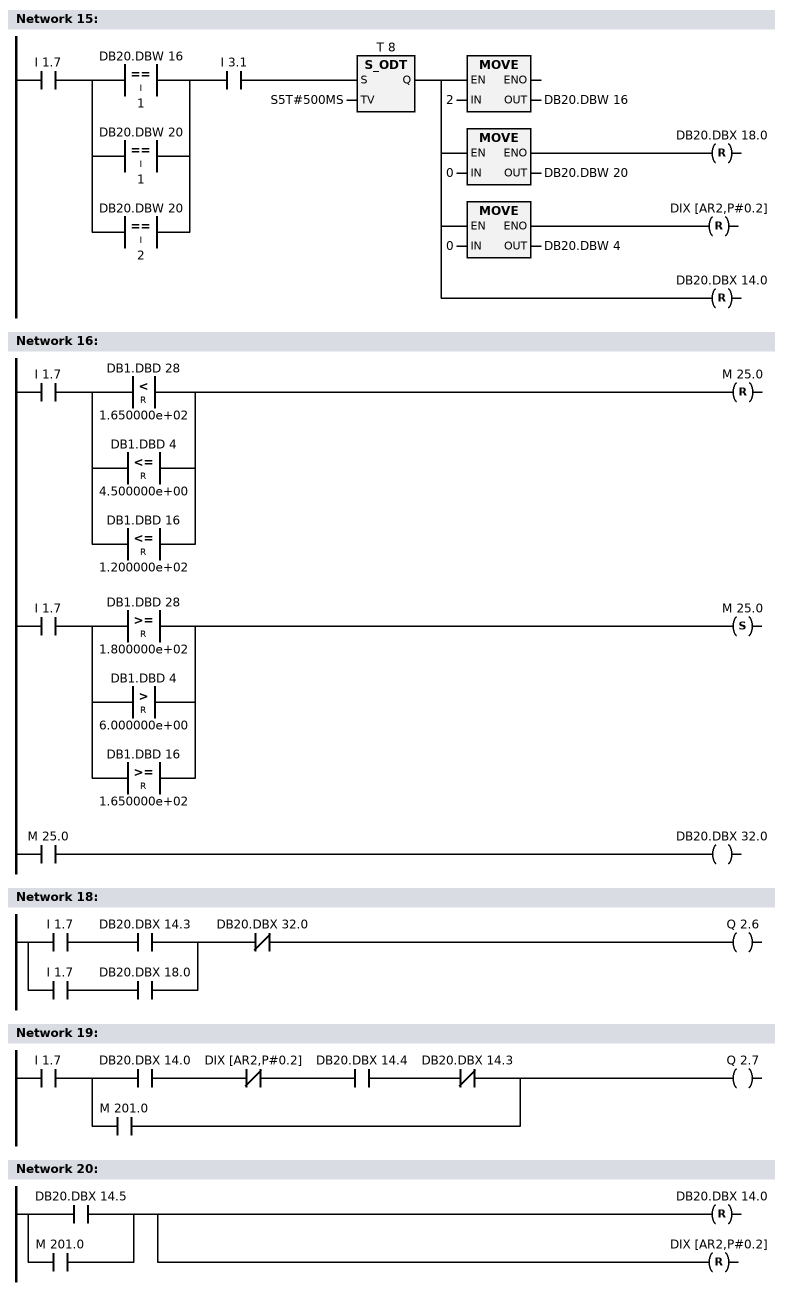
NETWORK
TITLE =
      A     I 1.7;
      A(;
      O(;
      L     DB20.DBW 16;
      L     1;
      ==I;
      );
      O(;
      L     DB20.DBW 20;
      L     1;
      ==I;
      );
      O(;
      L     DB20.DBW 20;
      L     2;
      ==I;
      );
      );
      A     I 3.1;
      L     S5T#500MS;
      SD    T 8;
      NOP   0;
      NOP   0;
      NOP   0;
      A     T 8;
      =     L 0.0;
      A     L 0.0;
      JNB   M016;
      L     2;
      T     DB20.DBW 16;
M016: NOP   0;
      A     L 0.0;
      JNB   M017;
      L     0;
      T     DB20.DBW 20;
      SET;
      SAVE;
      CLR;
M017: A     BR;
      R     DB20.DBX 18.0;
      A     L 0.0;
      JNB   M018;
      L     0;
      T     DB20.DBW 4;
      SET;
      SAVE;
      CLR;
M018: A     BR;
      R     DIX [AR2,P#0.2];
      A     L 0.0;
      BLD   102;
      R     DB20.DBX 14.0;
NETWORK
TITLE =
      A     I 1.7;
      A(;
      O(;
      L     DB1.DBD 28;
      L     1.650000e+02;
      <R;
      );
      O(;
      L     DB1.DBD 4;
      L     4.500000e+00;
      <=R;
      );
      O(;
      L     DB1.DBD 16;
      L     1.200000e+02;
      <=R;
      );
      );
      R     M 25.0;
      A     I 1.7;
      A(;
      O(;
      L     DB1.DBD 28;
      L     1.800000e+02;
      >=R;
      );
      O(;
      L     DB1.DBD 4;
      L     6.000000e+00;
      >R;
      );
      O(;
      L     DB1.DBD 16;
      L     1.650000e+02;
      >=R;
      );
      );
      S     M 25.0;
      A     M 25.0;
      =     DB20.DBX 32.0;
NETWORK
TITLE =
NETWORK
TITLE =
      A(;
      A     I 1.7;
      A     DB20.DBX 14.3;
      O;
      A     I 1.7;
      A     DB20.DBX 18.0;
      );
      AN    DB20.DBX 32.0;
      =     Q 2.6;
NETWORK
TITLE =
      A     I 1.7;
      A(;
      A     DB20.DBX 14.0;
      AN    DIX [AR2,P#0.2];
      A     DB20.DBX 14.4;
      AN    DB20.DBX 14.3;
      O     M 201.0;
      );
      =     Q 2.7;
NETWORK
TITLE =
      O     DB20.DBX 14.5;
      O     M 201.0;
      R     DB20.DBX 14.0;
      R     DIX [AR2,P#0.2];
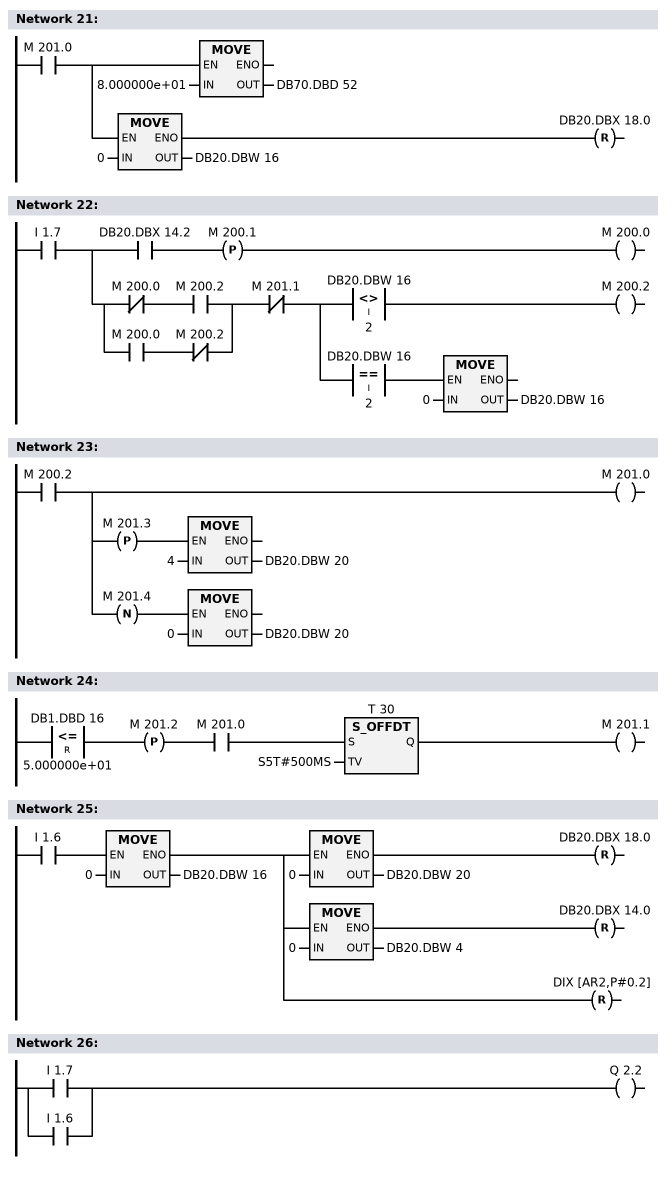
NETWORK
TITLE =
      A     M 201.0;
      =     L 0.0;
      A     L 0.0;
      JNB   M019;
      L     8.000000e+01;
      T     DB70.DBD 52;
M019: NOP   0;
      A     L 0.0;
      JNB   M020;
      L     0;
      T     DB20.DBW 16;
      SET;
      SAVE;
      CLR;
M020: A     BR;
      R     DB20.DBX 18.0;
NETWORK
TITLE =
      A     I 1.7;
      =     L 0.0;
      A     L 0.0;
      A     DB20.DBX 14.2;
      FP    M 200.1;
      =     M 200.0;
      A     L 0.0;
      A(;
      AN    M 200.0;
      A     M 200.2;
      O;
      A     M 200.0;
      AN    M 200.2;
      );
      AN    M 201.1;
      =     L 0.1;
      A     L 0.1;
      A(;
      L     DB20.DBW 16;
      L     2;
      <>I;
      );
      =     M 200.2;
      A     L 0.1;
      A(;
      L     DB20.DBW 16;
      L     2;
      ==I;
      );
      JNB   M021;
      L     0;
      T     DB20.DBW 16;
M021: NOP   0;
NETWORK
TITLE =
      A     M 200.2;
      =     L 0.0;
      A     L 0.0;
      BLD   102;
      =     M 201.0;
      A     L 0.0;
      FP    M 201.3;
      JNB   M022;
      L     4;
      T     DB20.DBW 20;
M022: NOP   0;
      A     L 0.0;
      FN    M 201.4;
      JNB   M023;
      L     0;
      T     DB20.DBW 20;
M023: NOP   0;
NETWORK
TITLE =
      A(;
      L     DB1.DBD 16;
      L     5.000000e+01;
      <=R;
      );
      FP    M 201.2;
      A     M 201.0;
      L     S5T#500MS;
      SF    T 30;
      NOP   0;
      NOP   0;
      NOP   0;
      A     T 30;
      =     M 201.1;
NETWORK
TITLE =
      A     I 1.6;
      JNB   M024;
      L     0;
      T     DB20.DBW 16;
      SET;
      SAVE;
      CLR;
M024: A     BR;
      =     L 0.0;
      A     L 0.0;
      JNB   M025;
      L     0;
      T     DB20.DBW 20;
      SET;
      SAVE;
      CLR;
M025: A     BR;
      R     DB20.DBX 18.0;
      A     L 0.0;
      JNB   M026;
      L     0;
      T     DB20.DBW 4;
      SET;
      SAVE;
      CLR;
M026: A     BR;
      R     DB20.DBX 14.0;
      A     L 0.0;
      BLD   102;
      R     DIX [AR2,P#0.2];
NETWORK
TITLE =
      O     I 1.7;
      O     I 1.6;
      =     Q 2.2;
